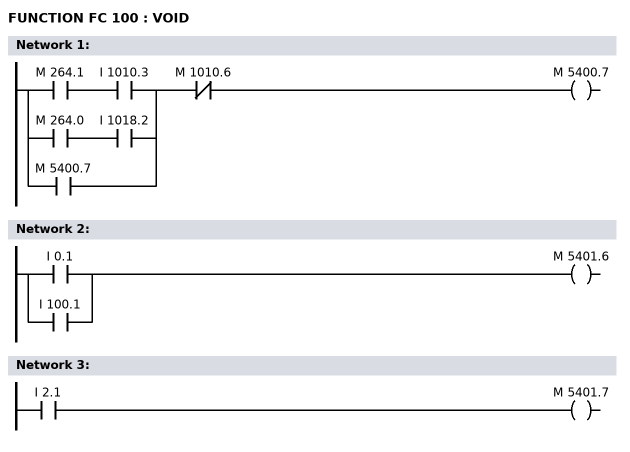

      A(    ;
      A     M    264.1;
      A     I   1010.3;
      O     ;
      A     M    264.0;
      A     I   1018.2;
      O     M   5400.7;
      )     ;
      AN    M   1010.6;
      =     M   5400.7;
NETWORK
TITLE =

      O     I      0.1;
      O     I    100.1;
      =     M   5401.6;
NETWORK
TITLE =

      A     I      2.1;
      =     M   5401.7;
NETWORK
TITLE =

      AN    OV;
      =     L      0.0;
      A     L      0.0;
      A     M   1003.7;
      AN    M   1000.0;
      A     M      0.5;
      =     M   5403.0;
      A     L      0.0;
      A     M   1003.7;
      A     M   1000.0;
      A     M      0.5;
      =     M   5403.1;
NETWORK
TITLE =

      AN    OV;
      =     L      0.0;
      A     L      0.0;
      A     M   1020.2;
      AN    I   1019.0;
      =     M   5403.2;
      A     L      0.0;
      A(    ;
      A     M   1020.2;
      A     I   1019.0;
      O     M   1035.1;
      )     ;
      =     M   5403.3;
NETWORK
TITLE =

      AN    OV;
      =     L      0.0;
      A     L      0.0;
      A     M   1008.2;
      AN    I   1011.0;
      =     M   5403.4;
      A     L      0.0;
      A(    ;
      A     M   1008.2;
      A     I   1011.0;
      O     M   1035.0;
      )     ;
      =     M   5403.5;
NETWORK
TITLE =
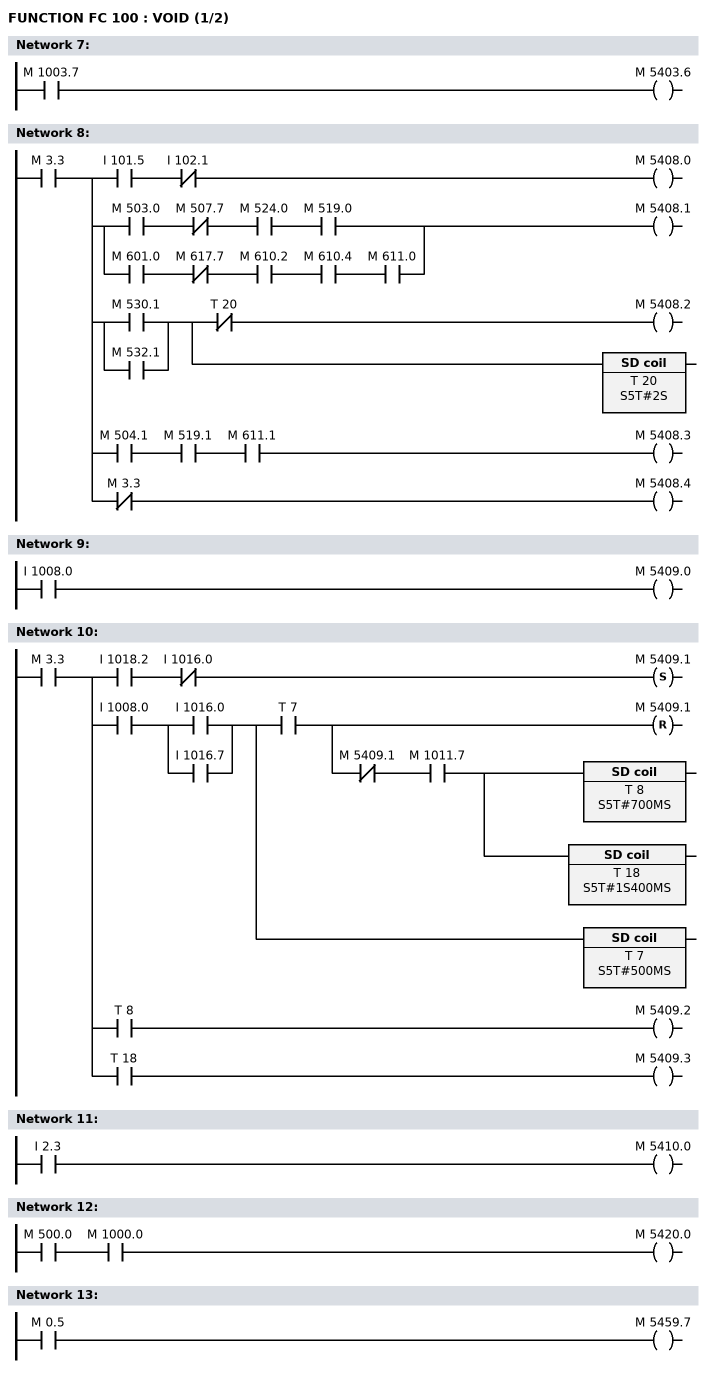

      A     M   1003.7;
      =     M   5403.6;
NETWORK
TITLE =

      A     M      3.3;
      =     L      0.0;
      A     L      0.0;
      A     I    101.5;
      AN    I    102.1;
      =     M   5408.0;
      A     L      0.0;
      A(    ;
      A     M    503.0;
      AN    M    507.7;
      A     M    524.0;
      A     M    519.0;
      O     ;
      A     M    601.0;
      AN    M    617.7;
      A     M    610.2;
      A     M    610.4;
      A     M    611.0;
      )     ;
      =     M   5408.1;
      A     L      0.0;
      A(    ;
      O     M    530.1;
      O     M    532.1;
      )     ;
      =     L      0.1;
      A     L      0.1;
      AN    T     20;
      =     M   5408.2;
      A     L      0.1;
      BLD   102;
      L     S5T#2S;
      SD    T     20;
      A     L      0.0;
      A     M    504.1;
      A     M    519.1;
      A     M    611.1;
      =     M   5408.3;
      A     L      0.0;
      AN    M      3.3;
      =     M   5408.4;
NETWORK
TITLE =

      A     I   1008.0;
      =     M   5409.0;
NETWORK
TITLE =

      A     M      3.3;
      =     L      0.0;
      A     L      0.0;
      A     I   1018.2;
      AN    I   1016.0;
      S     M   5409.1;
      A     L      0.0;
      A     I   1008.0;
      A(    ;
      O     I   1016.0;
      O     I   1016.7;
      )     ;
      =     L      0.1;
      A     L      0.1;
      A     T      7;
      =     L      0.2;
      A     L      0.2;
      BLD   102;
      R     M   5409.1;
      A     L      0.2;
      AN    M   5409.1;
      A     M   1011.7;
      L     S5T#700MS;
      SD    T      8;
      L     S5T#1S400MS;
      SD    T     18;
      A     L      0.1;
      BLD   102;
      L     S5T#500MS;
      SD    T      7;
      A     L      0.0;
      A     T      8;
      =     M   5409.2;
      A     L      0.0;
      A     T     18;
      =     M   5409.3;
NETWORK
TITLE =

      A     I      2.3;
      =     M   5410.0;
NETWORK
TITLE =

      A     M    500.0;
      A     M   1000.0;
      =     M   5420.0;
NETWORK
TITLE =

      A     M      0.5;
      =     M   5459.7;
NETWORK
TITLE =
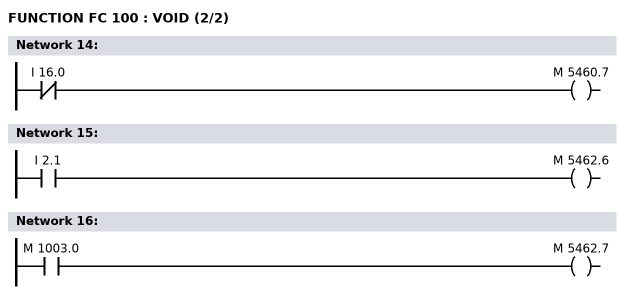

      AN    I     16.0;
      =     M   5460.7;
NETWORK
TITLE =

      A     I      2.1;
      =     M   5462.6;
NETWORK
TITLE =

      A     M   1003.0;
      =     M   5462.7;
NETWORK
TITLE =

      AN    OV;
      =     L      0.0;
      A     L      0.0;
      A(    ;
      ON    M    500.0;
      ON    I   1003.0;
      )     ;
      =     M   5463.0;
      A     L      0.0;
      A(    ;
      ON    M    500.6;
      ON    I   1000.4;
      )     ;
      =     M   5463.1;
      A     L      0.0;
      AN    M    516.0;
      AN    M    516.1;
      AN    M    516.2;
      AN    M    516.3;
      AN    M    516.4;
      AN    M    516.5;
      AN    M    516.6;
      AN    M    516.7;
      AN    M    517.1;
      AN    M    517.2;
      AN    M    517.3;
      AN    M   6060.0;
      AN    M    609.7;
      NOT   ;
      =     M   5463.2;
      A     L      0.0;
      A     M    517.0;
      =     M   5463.3;
      A     L      0.0;
      AN    M    541.0;
      AN    M    541.1;
      AN    M    543.0;
      NOT   ;
      =     M   5463.4;
      A     L      0.0;
      A     I    100.6;
      =     M   5463.5;
NETWORK
TITLE =

      AN    OV;
      =     L      0.0;
      A     L      0.0;
      AN    I   1011.0;
      =     M   5467.0;
      A     L      0.0;
      A     I   1011.1;
      =     M   5467.1;
      A     L      0.0;
      A     I   1011.2;
      =     M   5467.2;
      A     L      0.0;
      A     I   1011.4;
      =     M   5467.3;
      A     L      0.0;
      AN    M   1000.6;
      =     M   5467.4;
      A     L      0.0;
      A     I   1011.7;
      =     M   5467.6;
      A     L      0.0;
      A     M   1050.7;
      =     M   5467.7;
NETWORK
TITLE =
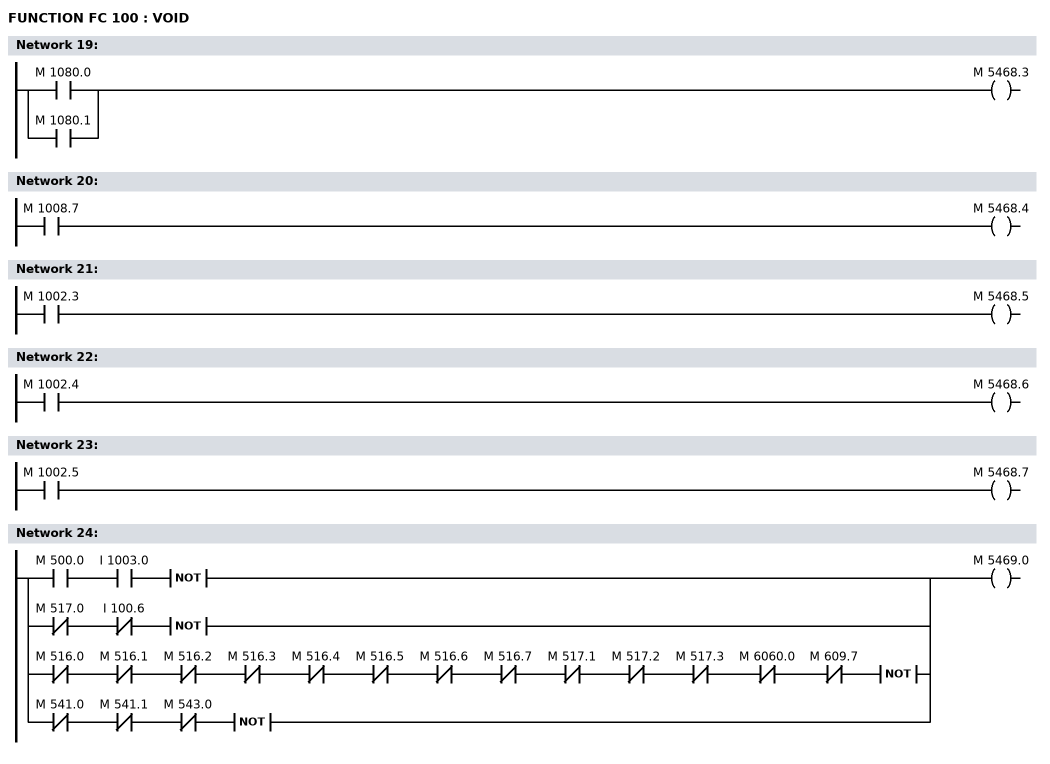

      O     M   1080.0;
      O     M   1080.1;
      =     M   5468.3;
NETWORK
TITLE =

      A     M   1008.7;
      =     M   5468.4;
NETWORK
TITLE =

      A     M   1002.3;
      =     M   5468.5;
NETWORK
TITLE =

      A     M   1002.4;
      =     M   5468.6;
NETWORK
TITLE =

      A     M   1002.5;
      =     M   5468.7;
NETWORK
TITLE =

      A     M    500.0;
      A     I   1003.0;
      NOT   ;
      O(    ;
      AN    M    517.0;
      AN    I    100.6;
      NOT   ;
      )     ;
      O(    ;
      AN    M    516.0;
      AN    M    516.1;
      AN    M    516.2;
      AN    M    516.3;
      AN    M    516.4;
      AN    M    516.5;
      AN    M    516.6;
      AN    M    516.7;
      AN    M    517.1;
      AN    M    517.2;
      AN    M    517.3;
      AN    M   6060.0;
      AN    M    609.7;
      NOT   ;
      )     ;
      O(    ;
      AN    M    541.0;
      AN    M    541.1;
      AN    M    543.0;
      NOT   ;
      )     ;
      =     M   5469.0;
END_FUNCTION

FUNCTION FC 101 : VOID
TITLE =
VERSION : 0.1

BEGIN
NETWORK
TITLE =
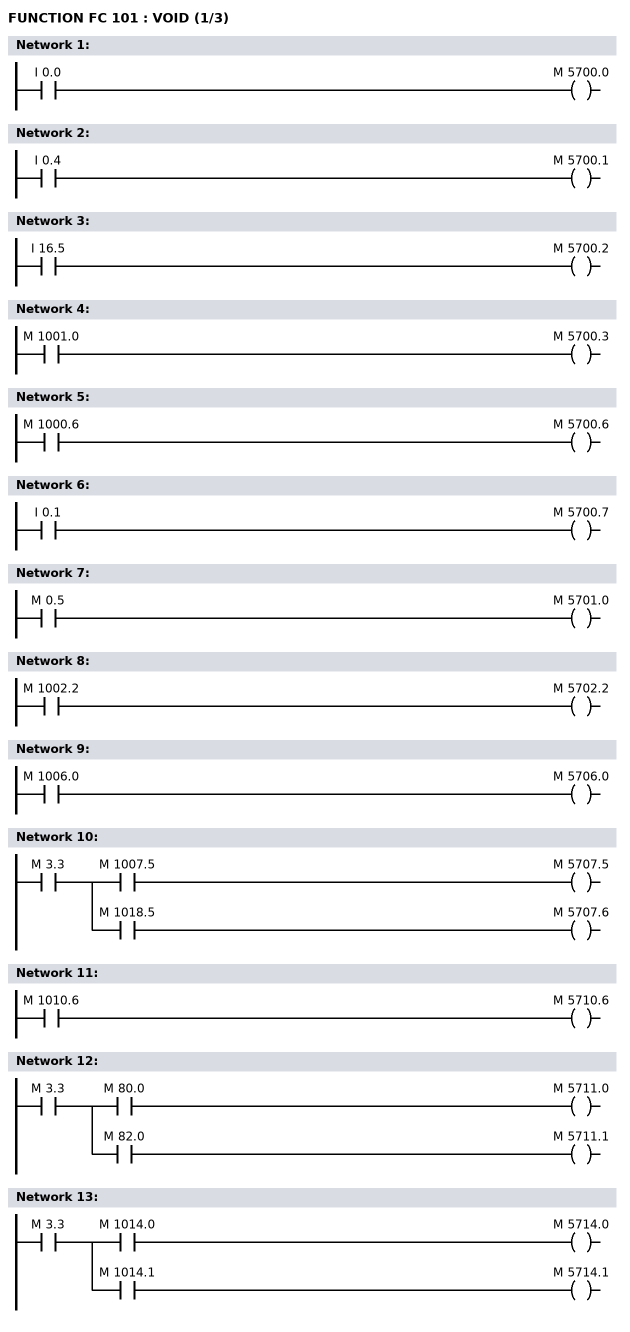

      A     I      0.0;
      =     M   5700.0;
NETWORK
TITLE =

      A     I      0.4;
      =     M   5700.1;
NETWORK
TITLE =

      A     I     16.5;
      =     M   5700.2;
NETWORK
TITLE =

      A     M   1001.0;
      =     M   5700.3;
NETWORK
TITLE =

      A     M   1000.6;
      =     M   5700.6;
NETWORK
TITLE =

      A     I      0.1;
      =     M   5700.7;
NETWORK
TITLE =

      A     M      0.5;
      =     M   5701.0;
NETWORK
TITLE =

      A     M   1002.2;
      =     M   5702.2;
NETWORK
TITLE =

      A     M   1006.0;
      =     M   5706.0;
NETWORK
TITLE =

      A     M      3.3;
      =     L      0.0;
      A     L      0.0;
      A     M   1007.5;
      =     M   5707.5;
      A     L      0.0;
      A     M   1018.5;
      =     M   5707.6;
NETWORK
TITLE =

      A     M   1010.6;
      =     M   5710.6;
NETWORK
TITLE =

      A     M      3.3;
      =     L      0.0;
      A     L      0.0;
      A     M     80.0;
      =     M   5711.0;
      A     L      0.0;
      A     M     82.0;
      =     M   5711.1;
NETWORK
TITLE =

      A     M      3.3;
      =     L      0.0;
      A     L      0.0;
      A     M   1014.0;
      =     M   5714.0;
      A     L      0.0;
      A     M   1014.1;
      =     M   5714.1;
NETWORK
TITLE =
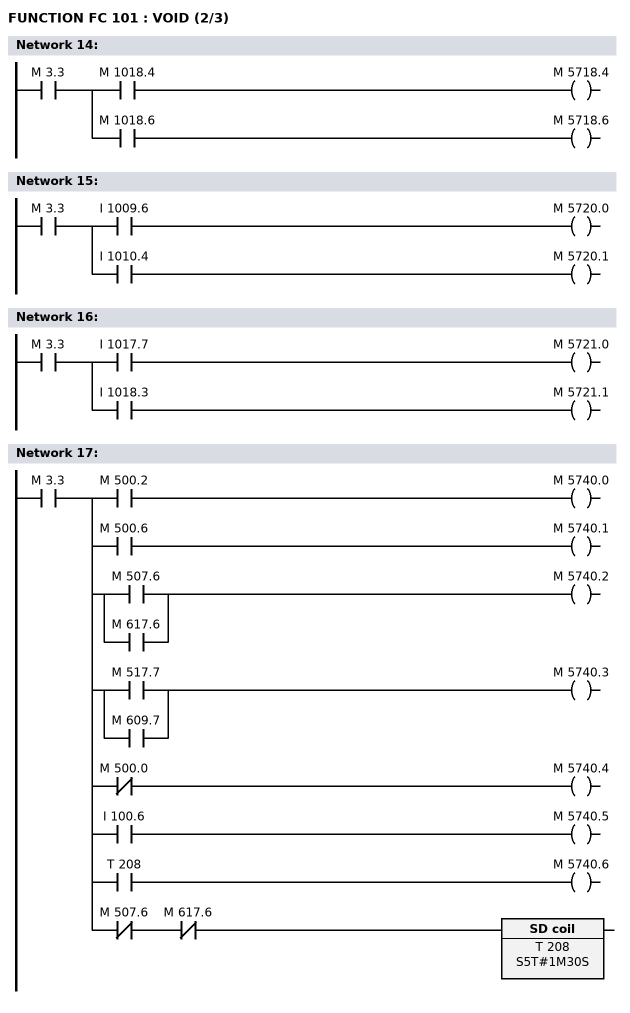

      A     M      3.3;
      =     L      0.0;
      A     L      0.0;
      A     M   1018.4;
      =     M   5718.4;
      A     L      0.0;
      A     M   1018.6;
      =     M   5718.6;
NETWORK
TITLE =

      A     M      3.3;
      =     L      0.0;
      A     L      0.0;
      A     I   1009.6;
      =     M   5720.0;
      A     L      0.0;
      A     I   1010.4;
      =     M   5720.1;
NETWORK
TITLE =

      A     M      3.3;
      =     L      0.0;
      A     L      0.0;
      A     I   1017.7;
      =     M   5721.0;
      A     L      0.0;
      A     I   1018.3;
      =     M   5721.1;
NETWORK
TITLE =

      A     M      3.3;
      =     L      0.0;
      A     L      0.0;
      A     M    500.2;
      =     M   5740.0;
      A     L      0.0;
      A     M    500.6;
      =     M   5740.1;
      A     L      0.0;
      A(    ;
      O     M    507.6;
      O     M    617.6;
      )     ;
      =     M   5740.2;
      A     L      0.0;
      A(    ;
      O     M    517.7;
      O     M    609.7;
      )     ;
      =     M   5740.3;
      A     L      0.0;
      AN    M    500.0;
      =     M   5740.4;
      A     L      0.0;
      A     I    100.6;
      =     M   5740.5;
      A     L      0.0;
      A     T    208;
      =     M   5740.6;
      A     L      0.0;
      AN    M    507.6;
      AN    M    617.6;
      L     S5T#1M30S;
      SD    T    208;
NETWORK
TITLE =
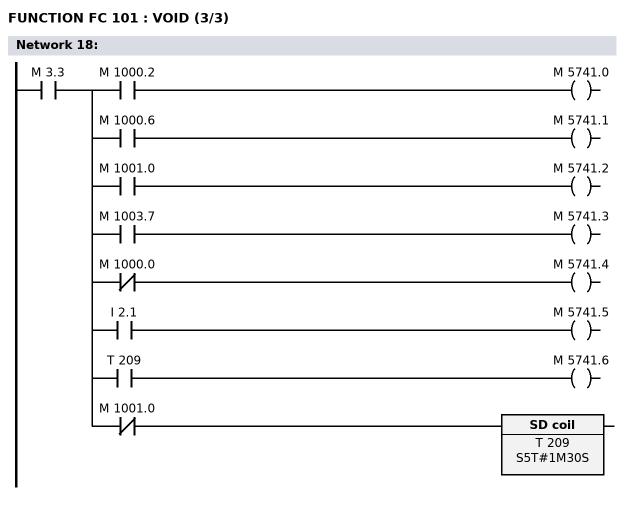

      A     M      3.3;
      =     L      0.0;
      A     L      0.0;
      A     M   1000.2;
      =     M   5741.0;
      A     L      0.0;
      A     M   1000.6;
      =     M   5741.1;
      A     L      0.0;
      A     M   1001.0;
      =     M   5741.2;
      A     L      0.0;
      A     M   1003.7;
      =     M   5741.3;
      A     L      0.0;
      AN    M   1000.0;
      =     M   5741.4;
      A     L      0.0;
      A     I      2.1;
      =     M   5741.5;
      A     L      0.0;
      A     T    209;
      =     M   5741.6;
      A     L      0.0;
      AN    M   1001.0;
      L     S5T#1M30S;
      SD    T    209;
END_FUNCTION

FUNCTION_BLOCK FB 105
TITLE =
VERSION : 0.1


VAR
  S711A_RBT1_WELD_OK_PLS : BOOL ;
  S711A_RBT1_WELD_NG_PLS : BOOL ;
  S711A_RBT1_WELD_PASS_PLS : BOOL ;
  S711A_CHECK_SUM_PLS : BOOL ;
  S711A_WELD_DATA_MOV_BUFF : BOOL ;
  MW_0_BUFF : ARRAY  [0 .. 59 ] OF WORD ;
  PLS1 : BOOL ;
  PLS2 : BOOL ;
END_VAR
VAR_TEMP
  SFC20_RET_VAL : INT ;
END_VAR
BEGIN
NETWORK
TITLE =MES 용접누락 DATA -> #711A차종코드(2011) 기준값 버퍼로 전송(LM)
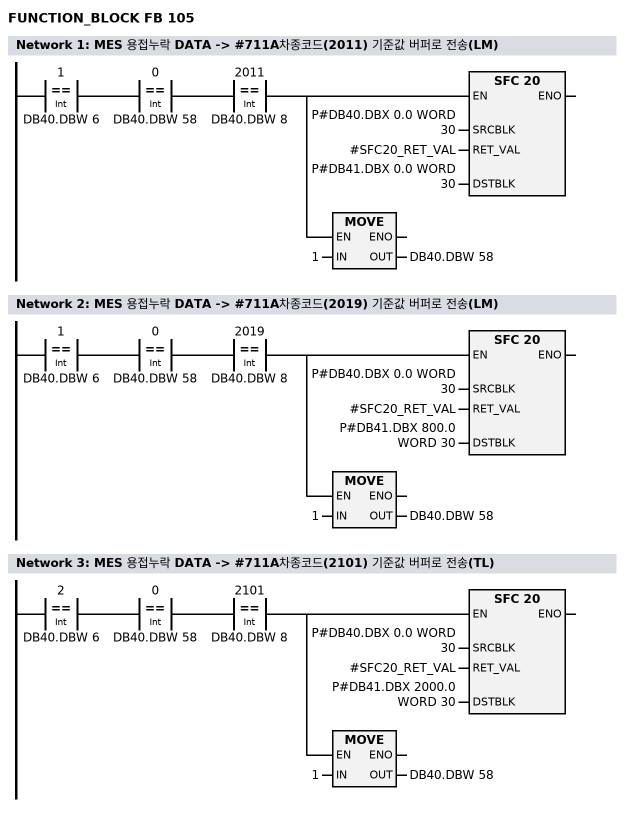

      A(    ;
      L     1;
      L     DB40.DBW    6;
      ==I   ;
      )     ;
      A(    ;
      L     0;
      L     DB40.DBW   58;
      ==I   ;
      )     ;
      A(    ;
      L     2011;
      L     DB40.DBW    8;
      ==I   ;
      )     ;
      =     L      2.0;
      A     L      2.0;
      JNB   _001;
      CALL SFC   20 (
           SRCBLK                   := P#DB40.DBX 0.0 WORD 30,
           RET_VAL                  := #SFC20_RET_VAL,
           DSTBLK                   := P#DB41.DBX 0.0 WORD 30);
_001: NOP   0;
      A     L      2.0;
      JNB   _002;
      L     1;
      T     DB40.DBW   58;
_002: NOP   0;
NETWORK
TITLE =MES 용접누락 DATA -> #711A차종코드(2019) 기준값 버퍼로 전송(LM)

      A(    ;
      L     1;
      L     DB40.DBW    6;
      ==I   ;
      )     ;
      A(    ;
      L     0;
      L     DB40.DBW   58;
      ==I   ;
      )     ;
      A(    ;
      L     2019;
      L     DB40.DBW    8;
      ==I   ;
      )     ;
      =     L      2.0;
      A     L      2.0;
      JNB   _003;
      CALL SFC   20 (
           SRCBLK                   := P#DB40.DBX 0.0 WORD 30,
           RET_VAL                  := #SFC20_RET_VAL,
           DSTBLK                   := P#DB41.DBX 800.0 WORD 30);
_003: NOP   0;
      A     L      2.0;
      JNB   _004;
      L     1;
      T     DB40.DBW   58;
_004: NOP   0;
NETWORK
TITLE =MES 용접누락 DATA -> #711A차종코드(2101) 기준값 버퍼로 전송(TL)

      A(    ;
      L     2;
      L     DB40.DBW    6;
      ==I   ;
      )     ;
      A(    ;
      L     0;
      L     DB40.DBW   58;
      ==I   ;
      )     ;
      A(    ;
      L     2101;
      L     DB40.DBW    8;
      ==I   ;
      )     ;
      =     L      2.0;
      A     L      2.0;
      JNB   _005;
      CALL SFC   20 (
           SRCBLK                   := P#DB40.DBX 0.0 WORD 30,
           RET_VAL                  := #SFC20_RET_VAL,
           DSTBLK                   := P#DB41.DBX 2000.0 WORD 30);
_005: NOP   0;
      A     L      2.0;
      JNB   _006;
      L     1;
      T     DB40.DBW   58;
_006: NOP   0;
NETWORK
TITLE =#711A-2 RBT1호 용접카운터 INT -> DB로 전송보조

      AN    OV;
      =     L      2.0;
      A     L      2.0;
      A     I   1004.0;
      =     M     11.0;
      A     L      2.0;
      A     I   1004.1;
      =     M     11.1;
      A     L      2.0;
      A     I   1004.2;
      =     M     11.2;
      A     L      2.0;
      A     I   1004.3;
      =     M     11.3;
      A     L      2.0;
      A     I   1004.4;
      =     M     11.4;
      A     L      2.0;
      AN    M      3.3;
      =     L      2.1;
      A     L      2.1;
      A     I   1004.5;
      =     M     11.5;
      A     L      2.1;
      A     I   1004.6;
      =     M     11.6;
      A     L      2.1;
      A     I   1004.7;
      =     M     11.7;
      A     L      2.0;
      AN    I    102.1;
      A     I   1000.1;
      S     M    531.7;
      A     L      2.0;
      AN    I    102.1;
      A     M    505.1;
      A     M    540.1;
      A     M    540.7;
      R     M    531.7;
NETWORK
TITLE =#711A-2 RBT1호 용접카운터 INT -> DB로 전송
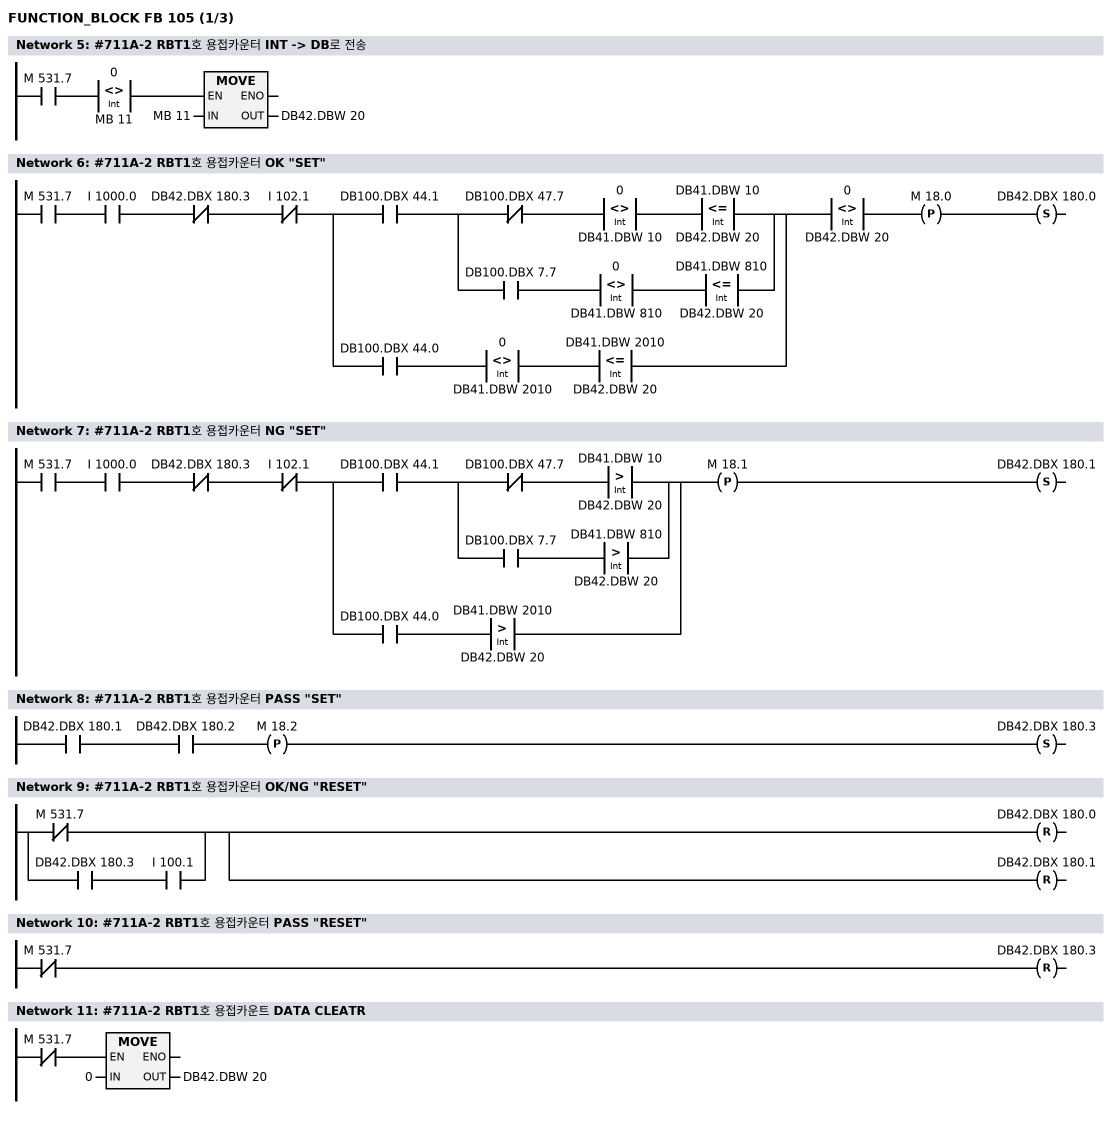

      A     M    531.7;
      A(    ;
      L     0;
      L     MB    11;
      <>I   ;
      )     ;
      JNB   _007;
      L     MB    11;
      T     DB42.DBW   20;
_007: NOP   0;
NETWORK
TITLE =#711A-2 RBT1호 용접카운터 OK "SET"

      A     M    531.7;
      A     I   1000.0;
      AN    DB42.DBX  180.3;
      AN    I    102.1;
      A(    ;
      A     DB100.DBX   44.1;
      A(    ;
      AN    DB100.DBX   47.7;
      A(    ;
      L     0;
      L     DB41.DBW   10;
      <>I   ;
      )     ;
      A(    ;
      L     DB41.DBW   10;
      L     DB42.DBW   20;
      <=I   ;
      )     ;
      O     ;
      A     DB100.DBX    7.7;
      A(    ;
      L     0;
      L     DB41.DBW  810;
      <>I   ;
      )     ;
      A(    ;
      L     DB41.DBW  810;
      L     DB42.DBW   20;
      <=I   ;
      )     ;
      )     ;
      O     ;
      A     DB100.DBX   44.0;
      A(    ;
      L     0;
      L     DB41.DBW 2010;
      <>I   ;
      )     ;
      A(    ;
      L     DB41.DBW 2010;
      L     DB42.DBW   20;
      <=I   ;
      )     ;
      )     ;
      A(    ;
      L     0;
      L     DB42.DBW   20;
      <>I   ;
      )     ;
      FP    M     18.0;
      S     DB42.DBX  180.0;
NETWORK
TITLE =#711A-2 RBT1호 용접카운터 NG "SET"

      A     M    531.7;
      A     I   1000.0;
      AN    DB42.DBX  180.3;
      AN    I    102.1;
      A(    ;
      A     DB100.DBX   44.1;
      A(    ;
      AN    DB100.DBX   47.7;
      A(    ;
      L     DB41.DBW   10;
      L     DB42.DBW   20;
      >I    ;
      )     ;
      O     ;
      A     DB100.DBX    7.7;
      A(    ;
      L     DB41.DBW  810;
      L     DB42.DBW   20;
      >I    ;
      )     ;
      )     ;
      O     ;
      A     DB100.DBX   44.0;
      A(    ;
      L     DB41.DBW 2010;
      L     DB42.DBW   20;
      >I    ;
      )     ;
      )     ;
      FP    M     18.1;
      S     DB42.DBX  180.1;
NETWORK
TITLE =#711A-2 RBT1호 용접카운터 PASS "SET"

      A     DB42.DBX  180.1;
      A     DB42.DBX  180.2;
      FP    M     18.2;
      S     DB42.DBX  180.3;
NETWORK
TITLE =#711A-2 RBT1호 용접카운터 OK/NG "RESET"

      ON    M    531.7;
      O     ;
      A     DB42.DBX  180.3;
      A     I    100.1;
      R     DB42.DBX  180.0;
      R     DB42.DBX  180.1;
NETWORK
TITLE =#711A-2 RBT1호 용접카운터 PASS "RESET"

      AN    M    531.7;
      R     DB42.DBX  180.3;
NETWORK
TITLE =#711A-2 RBT1호 용접카운트 DATA CLEATR

      AN    M    531.7;
      JNB   _008;
      L     0;
      T     DB42.DBW   20;
_008: NOP   0;
NETWORK
TITLE =#711A-2 RBT1호 용접DATA 관련(공정 및 차종정보)
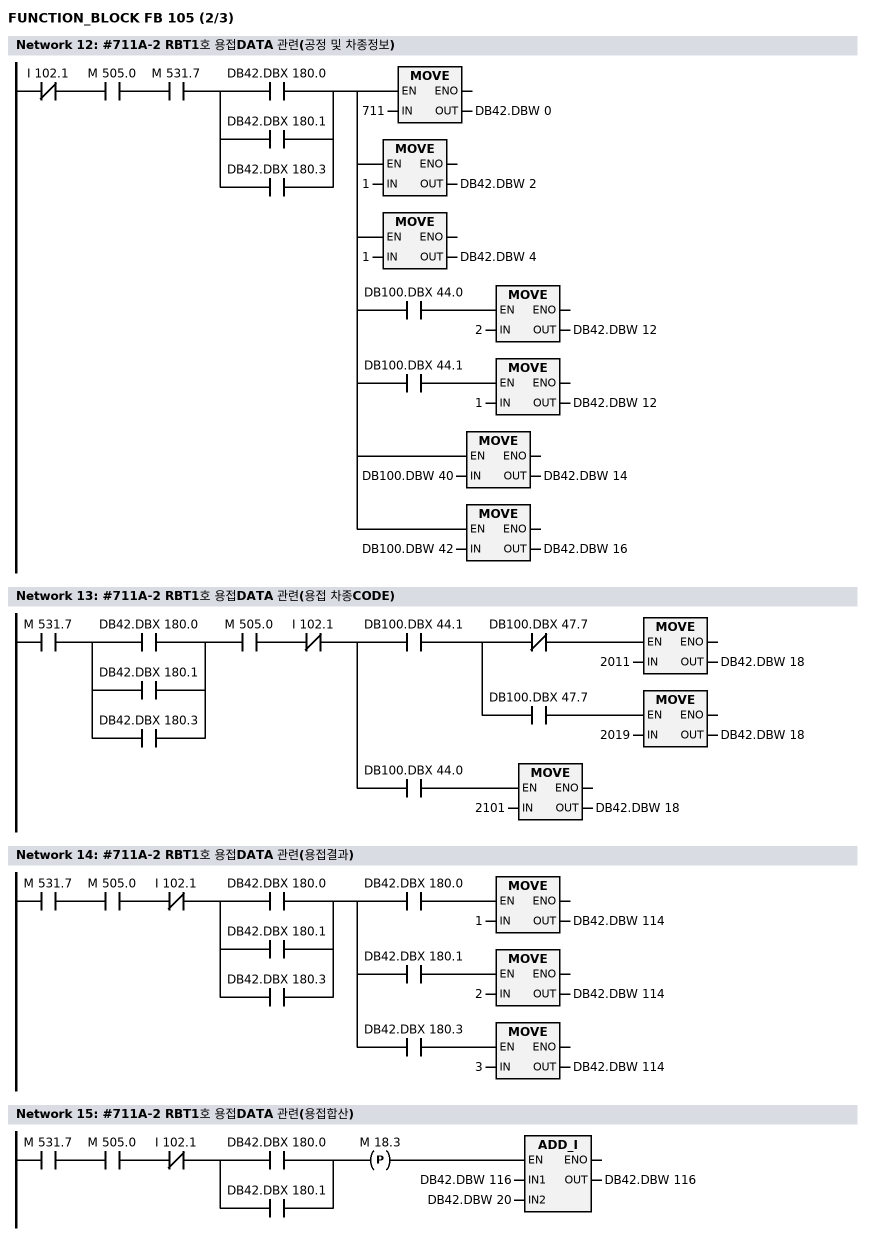

      AN    I    102.1;
      A     M    505.0;
      A     M    531.7;
      A(    ;
      O     DB42.DBX  180.0;
      O     DB42.DBX  180.1;
      O     DB42.DBX  180.3;
      )     ;
      =     L      2.0;
      A     L      2.0;
      JNB   _009;
      L     711;
      T     DB42.DBW    0;
_009: NOP   0;
      A     L      2.0;
      JNB   _00a;
      L     1;
      T     DB42.DBW    2;
_00a: NOP   0;
      A     L      2.0;
      JNB   _00b;
      L     1;
      T     DB42.DBW    4;
_00b: NOP   0;
      A     L      2.0;
      A     DB100.DBX   44.0;
      JNB   _00c;
      L     2;
      T     DB42.DBW   12;
_00c: NOP   0;
      A     L      2.0;
      A     DB100.DBX   44.1;
      JNB   _00d;
      L     1;
      T     DB42.DBW   12;
_00d: NOP   0;
      A     L      2.0;
      JNB   _00e;
      L     DB100.DBW   40;
      T     DB42.DBW   14;
_00e: NOP   0;
      A     L      2.0;
      JNB   _00f;
      L     DB100.DBW   42;
      T     DB42.DBW   16;
_00f: NOP   0;
NETWORK
TITLE =#711A-2 RBT1호 용접DATA 관련(용접 차종CODE)

      A     M    531.7;
      A(    ;
      O     DB42.DBX  180.0;
      O     DB42.DBX  180.1;
      O     DB42.DBX  180.3;
      )     ;
      A     M    505.0;
      AN    I    102.1;
      =     L      2.0;
      A     L      2.0;
      A     DB100.DBX   44.1;
      =     L      2.1;
      A     L      2.1;
      AN    DB100.DBX   47.7;
      JNB   _010;
      L     2011;
      T     DB42.DBW   18;
_010: NOP   0;
      A     L      2.1;
      A     DB100.DBX   47.7;
      JNB   _011;
      L     2019;
      T     DB42.DBW   18;
_011: NOP   0;
      A     L      2.0;
      A     DB100.DBX   44.0;
      JNB   _012;
      L     2101;
      T     DB42.DBW   18;
_012: NOP   0;
NETWORK
TITLE =#711A-2 RBT1호 용접DATA 관련(용접결과)

      A     M    531.7;
      A     M    505.0;
      AN    I    102.1;
      A(    ;
      O     DB42.DBX  180.0;
      O     DB42.DBX  180.1;
      O     DB42.DBX  180.3;
      )     ;
      =     L      2.0;
      A     L      2.0;
      A     DB42.DBX  180.0;
      JNB   _013;
      L     1;
      T     DB42.DBW  114;
_013: NOP   0;
      A     L      2.0;
      A     DB42.DBX  180.1;
      JNB   _014;
      L     2;
      T     DB42.DBW  114;
_014: NOP   0;
      A     L      2.0;
      A     DB42.DBX  180.3;
      JNB   _015;
      L     3;
      T     DB42.DBW  114;
_015: NOP   0;
NETWORK
TITLE =#711A-2 RBT1호 용접DATA 관련(용접합산)

      A     M    531.7;
      A     M    505.0;
      AN    I    102.1;
      A(    ;
      O     DB42.DBX  180.0;
      O     DB42.DBX  180.1;
      )     ;
      FP    M     18.3;
      JNB   _016;
      L     DB42.DBW  116;
      L     DB42.DBW   20;
      +I    ;
      T     DB42.DBW  116;
_016: NOP   0;
NETWORK
TITLE =용접누락버퍼로 공정DATA 전송
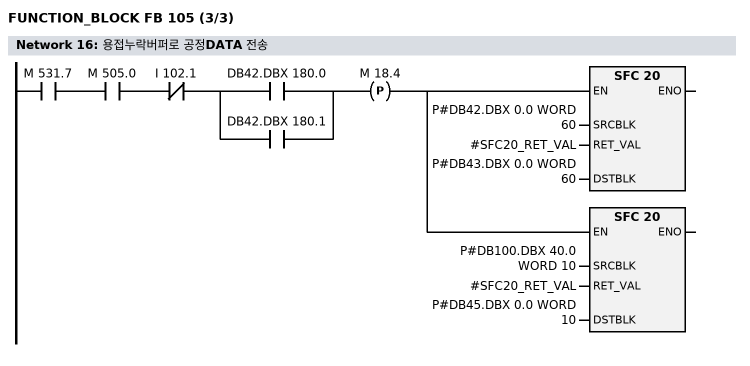

      A     M    531.7;
      A     M    505.0;
      AN    I    102.1;
      A(    ;
      O     DB42.DBX  180.0;
      O     DB42.DBX  180.1;
      )     ;
      FP    M     18.4;
      =     L      2.0;
      A     L      2.0;
      JNB   _017;
      CALL SFC   20 (
           SRCBLK                   := P#DB42.DBX 0.0 WORD 60,
           RET_VAL                  := #SFC20_RET_VAL,
           DSTBLK                   := P#DB43.DBX 0.0 WORD 60);
_017: NOP   0;
      A     L      2.0;
      JNB   _018;
      CALL SFC   20 (
           SRCBLK                   := P#DB100.DBX 40.0 WORD 10,
           RET_VAL                  := #SFC20_RET_VAL,
           DSTBLK                   := P#DB45.DBX 0.0 WORD 10);
_018: NOP   0;
NETWORK
TITLE =용접누락버퍼로 공정DATA 전송

      AN    M    531.7;
      FP    M     18.5;
      =     L      2.0;
      A(    ;
      A     L      2.0;
      JNB   _019;
      CALL SFC   20 (
           SRCBLK                   := P#DB43.DBX 960.0 WORD 60,
           RET_VAL                  := #SFC20_RET_VAL,
           DSTBLK                   := P#DB43.DBX 1080.0 WORD 60);
_019: A     BR;
      )     ;
      JNB   _01a;
      CALL SFC   20 (
           SRCBLK                   := P#DB43.DBX 840.0 WORD 60,
           RET_VAL                  := #SFC20_RET_VAL,
           DSTBLK                   := P#DB43.DBX 960.0 WORD 60);
_01a: NOP   0;
      A(    ;
      A     L      2.0;
      JNB   _01b;
      CALL SFC   20 (
           SRCBLK                   := P#DB43.DBX 720.0 WORD 60,
           RET_VAL                  := #SFC20_RET_VAL,
           DSTBLK                   := P#DB43.DBX 840.0 WORD 60);
_01b: A     BR;
      )     ;
      JNB   _01c;
      CALL SFC   20 (
           SRCBLK                   := P#DB43.DBX 600.0 WORD 60,
           RET_VAL                  := #SFC20_RET_VAL,
           DSTBLK                   := P#DB43.DBX 720.0 WORD 60);
_01c: NOP   0;
      A(    ;
      A     L      2.0;
      JNB   _01d;
      CALL SFC   20 (
           SRCBLK                   := P#DB43.DBX 480.0 WORD 60,
           RET_VAL                  := #SFC20_RET_VAL,
           DSTBLK                   := P#DB43.DBX 600.0 WORD 60);
_01d: A     BR;
      )     ;
      JNB   _01e;
      CALL SFC   20 (
           SRCBLK                   := P#DB43.DBX 360.0 WORD 60,
           RET_VAL                  := #SFC20_RET_VAL,
           DSTBLK                   := P#DB43.DBX 480.0 WORD 60);
_01e: NOP   0;
      A(    ;
      A     L      2.0;
      JNB   _01f;
      CALL SFC   20 (
           SRCBLK                   := P#DB43.DBX 240.0 WORD 60,
           RET_VAL                  := #SFC20_RET_VAL,
           DSTBLK                   := P#DB43.DBX 360.0 WORD 60);
_01f: A     BR;
      )     ;
      JNB   _020;
      CALL SFC   20 (
           SRCBLK                   := P#DB43.DBX 120.0 WORD 60,
           RET_VAL                  := #SFC20_RET_VAL,
           DSTBLK                   := P#DB43.DBX 240.0 WORD 60);
_020: NOP   0;
      A     L      2.0;
      JNB   _021;
      CALL SFC   20 (
           SRCBLK                   := P#DB43.DBX 0.0 WORD 60,
           RET_VAL                  := #SFC20_RET_VAL,
           DSTBLK                   := P#DB43.DBX 120.0 WORD 60);
_021: NOP   0;
      A     L      2.0;
      JNB   _022;
      CALL SFC   21 (
           BVAL                     := P#M 30.0 WORD 1,
           RET_VAL                  := #SFC20_RET_VAL,
           BLK                      := P#DB43.DBX 0.0 WORD 60);
_022: NOP   0;
      A(    ;
      A     L      2.0;
      JNB   _023;
      CALL SFC   20 (
           SRCBLK                   := P#DB45.DBX 160.0 WORD 10,
           RET_VAL                  := #SFC20_RET_VAL,
           DSTBLK                   := P#DB45.DBX 180.0 WORD 10);
_023: A     BR;
      )     ;
      JNB   _024;
      CALL SFC   20 (
           SRCBLK                   := P#DB45.DBX 140.0 WORD 10,
           RET_VAL                  := #SFC20_RET_VAL,
           DSTBLK                   := P#DB45.DBX 160.0 WORD 10);
_024: NOP   0;
      A(    ;
      A     L      2.0;
      JNB   _025;
      CALL SFC   20 (
           SRCBLK                   := P#DB45.DBX 120.0 WORD 10,
           RET_VAL                  := #SFC20_RET_VAL,
           DSTBLK                   := P#DB45.DBX 140.0 WORD 10);
_025: A     BR;
      )     ;
      JNB   _026;
      CALL SFC   20 (
           SRCBLK                   := P#DB45.DBX 100.0 WORD 10,
           RET_VAL                  := #SFC20_RET_VAL,
           DSTBLK                   := P#DB45.DBX 120.0 WORD 10);
_026: NOP   0;
      A(    ;
      A     L      2.0;
      JNB   _027;
      CALL SFC   20 (
           SRCBLK                   := P#DB45.DBX 80.0 WORD 10,
           RET_VAL                  := #SFC20_RET_VAL,
           DSTBLK                   := P#DB45.DBX 100.0 WORD 10);
_027: A     BR;
      )     ;
      JNB   _028;
      CALL SFC   20 (
           SRCBLK                   := P#DB45.DBX 60.0 WORD 10,
           RET_VAL                  := #SFC20_RET_VAL,
           DSTBLK                   := P#DB45.DBX 80.0 WORD 10);
_028: NOP   0;
      A(    ;
      A     L      2.0;
      JNB   _029;
      CALL SFC   20 (
           SRCBLK                   := P#DB45.DBX 40.0 WORD 10,
           RET_VAL                  := #SFC20_RET_VAL,
           DSTBLK                   := P#DB45.DBX 60.0 WORD 10);
_029: A     BR;
      )     ;
      JNB   _02a;
      CALL SFC   20 (
           SRCBLK                   := P#DB45.DBX 20.0 WORD 10,
           RET_VAL                  := #SFC20_RET_VAL,
           DSTBLK                   := P#DB45.DBX 40.0 WORD 10);
_02a: NOP   0;
      A     L      2.0;
      JNB   _02b;
      CALL SFC   20 (
           SRCBLK                   := P#DB45.DBX 0.0 WORD 10,
           RET_VAL                  := #SFC20_RET_VAL,
           DSTBLK                   := P#DB45.DBX 20.0 WORD 10);
_02b: NOP   0;
      A     L      2.0;
      JNB   _02c;
      CALL SFC   21 (
           BVAL                     := P#M 30.0 WORD 1,
           RET_VAL                  := #SFC20_RET_VAL,
           BLK                      := P#DB45.DBX 0.0 WORD 10);
_02c: NOP   0;
NETWORK
TITLE =용접누락버퍼로 공정DATA 전송
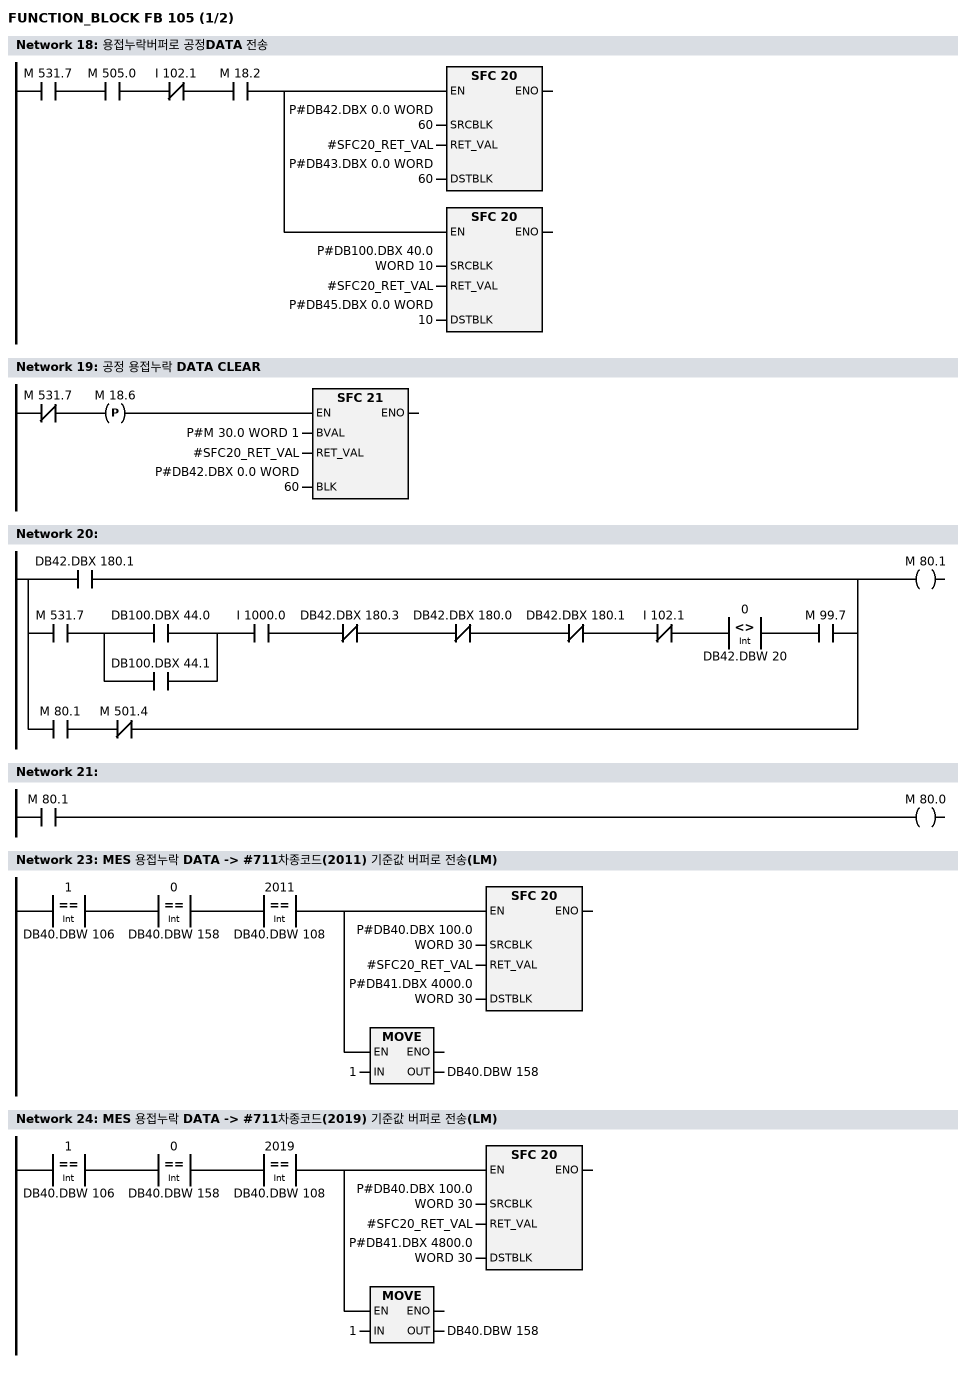

      A     M    531.7;
      A     M    505.0;
      AN    I    102.1;
      A     M     18.2;
      =     L      2.0;
      A     L      2.0;
      JNB   _02d;
      CALL SFC   20 (
           SRCBLK                   := P#DB42.DBX 0.0 WORD 60,
           RET_VAL                  := #SFC20_RET_VAL,
           DSTBLK                   := P#DB43.DBX 0.0 WORD 60);
_02d: NOP   0;
      A     L      2.0;
      JNB   _02e;
      CALL SFC   20 (
           SRCBLK                   := P#DB100.DBX 40.0 WORD 10,
           RET_VAL                  := #SFC20_RET_VAL,
           DSTBLK                   := P#DB45.DBX 0.0 WORD 10);
_02e: NOP   0;
NETWORK
TITLE =공정 용접누락 DATA CLEAR

      AN    M    531.7;
      FP    M     18.6;
      JNB   _02f;
      CALL SFC   21 (
           BVAL                     := P#M 30.0 WORD 1,
           RET_VAL                  := #SFC20_RET_VAL,
           BLK                      := P#DB42.DBX 0.0 WORD 60);
_02f: NOP   0;
NETWORK
TITLE =

      O     DB42.DBX  180.1;
      O     ;
      A     M    531.7;
      A(    ;
      O     DB100.DBX   44.0;
      O     DB100.DBX   44.1;
      )     ;
      A     I   1000.0;
      AN    DB42.DBX  180.3;
      AN    DB42.DBX  180.0;
      AN    DB42.DBX  180.1;
      AN    I    102.1;
      A(    ;
      L     0;
      L     DB42.DBW   20;
      <>I   ;
      )     ;
      A     M     99.7;
      O     ;
      A     M     80.1;
      AN    M    501.4;
      =     M     80.1;
NETWORK
TITLE =

      A     M     80.1;
      =     M     80.0;
NETWORK
TITLE =

NETWORK
TITLE =MES 용접누락 DATA -> #711차종코드(2011) 기준값 버퍼로 전송(LM)

      A(    ;
      L     1;
      L     DB40.DBW  106;
      ==I   ;
      )     ;
      A(    ;
      L     0;
      L     DB40.DBW  158;
      ==I   ;
      )     ;
      A(    ;
      L     2011;
      L     DB40.DBW  108;
      ==I   ;
      )     ;
      =     L      2.0;
      A     L      2.0;
      JNB   _030;
      CALL SFC   20 (
           SRCBLK                   := P#DB40.DBX 100.0 WORD 30,
           RET_VAL                  := #SFC20_RET_VAL,
           DSTBLK                   := P#DB41.DBX 4000.0 WORD 30);
_030: NOP   0;
      A     L      2.0;
      JNB   _031;
      L     1;
      T     DB40.DBW  158;
_031: NOP   0;
NETWORK
TITLE =MES 용접누락 DATA -> #711차종코드(2019) 기준값 버퍼로 전송(LM)

      A(    ;
      L     1;
      L     DB40.DBW  106;
      ==I   ;
      )     ;
      A(    ;
      L     0;
      L     DB40.DBW  158;
      ==I   ;
      )     ;
      A(    ;
      L     2019;
      L     DB40.DBW  108;
      ==I   ;
      )     ;
      =     L      2.0;
      A     L      2.0;
      JNB   _032;
      CALL SFC   20 (
           SRCBLK                   := P#DB40.DBX 100.0 WORD 30,
           RET_VAL                  := #SFC20_RET_VAL,
           DSTBLK                   := P#DB41.DBX 4800.0 WORD 30);
_032: NOP   0;
      A     L      2.0;
      JNB   _033;
      L     1;
      T     DB40.DBW  158;
_033: NOP   0;
NETWORK
TITLE =MES 용접누락 DATA -> #711차종코드(2101) 기준값 버퍼로 전송(TL)
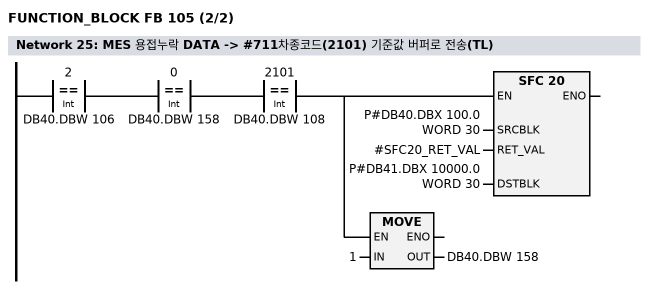

      A(    ;
      L     2;
      L     DB40.DBW  106;
      ==I   ;
      )     ;
      A(    ;
      L     0;
      L     DB40.DBW  158;
      ==I   ;
      )     ;
      A(    ;
      L     2101;
      L     DB40.DBW  108;
      ==I   ;
      )     ;
      =     L      2.0;
      A     L      2.0;
      JNB   _034;
      CALL SFC   20 (
           SRCBLK                   := P#DB40.DBX 100.0 WORD 30,
           RET_VAL                  := #SFC20_RET_VAL,
           DSTBLK                   := P#DB41.DBX 10000.0 WORD 30);
_034: NOP   0;
      A     L      2.0;
      JNB   _035;
      L     1;
      T     DB40.DBW  158;
_035: NOP   0;
NETWORK
TITLE =#711 RBT2호 용접카운터 INT -> DB로 전송보조

      AN    OV;
      =     L      2.0;
      A     L      2.0;
      A     I   1020.0;
      =     M     15.0;
      A     L      2.0;
      A     I   1020.1;
      =     M     15.1;
      A     L      2.0;
      A     I   1020.2;
      =     M     15.2;
      A     L      2.0;
      A     I   1020.3;
      =     M     15.3;
      A     L      2.0;
      A     I   1020.4;
      =     M     15.4;
      A     L      2.0;
      AN    M      3.3;
      =     L      2.1;
      A     L      2.1;
      A     I   1020.5;
      =     M     15.5;
      A     L      2.1;
      A     I   1020.6;
      =     M     15.6;
      A     L      2.1;
      A     I   1020.7;
      =     M     15.7;
      A     L      2.0;
      A     I   1016.1;
      S     M     16.7;
      A     L      2.0;
      A(    ;
      A     M   1010.7;
      A     M   1002.1;
      O     M   4712.1;
      )     ;
      R     M     16.7;
NETWORK
TITLE =#711 RBT2호 용접카운터 INT -> DB로 전송
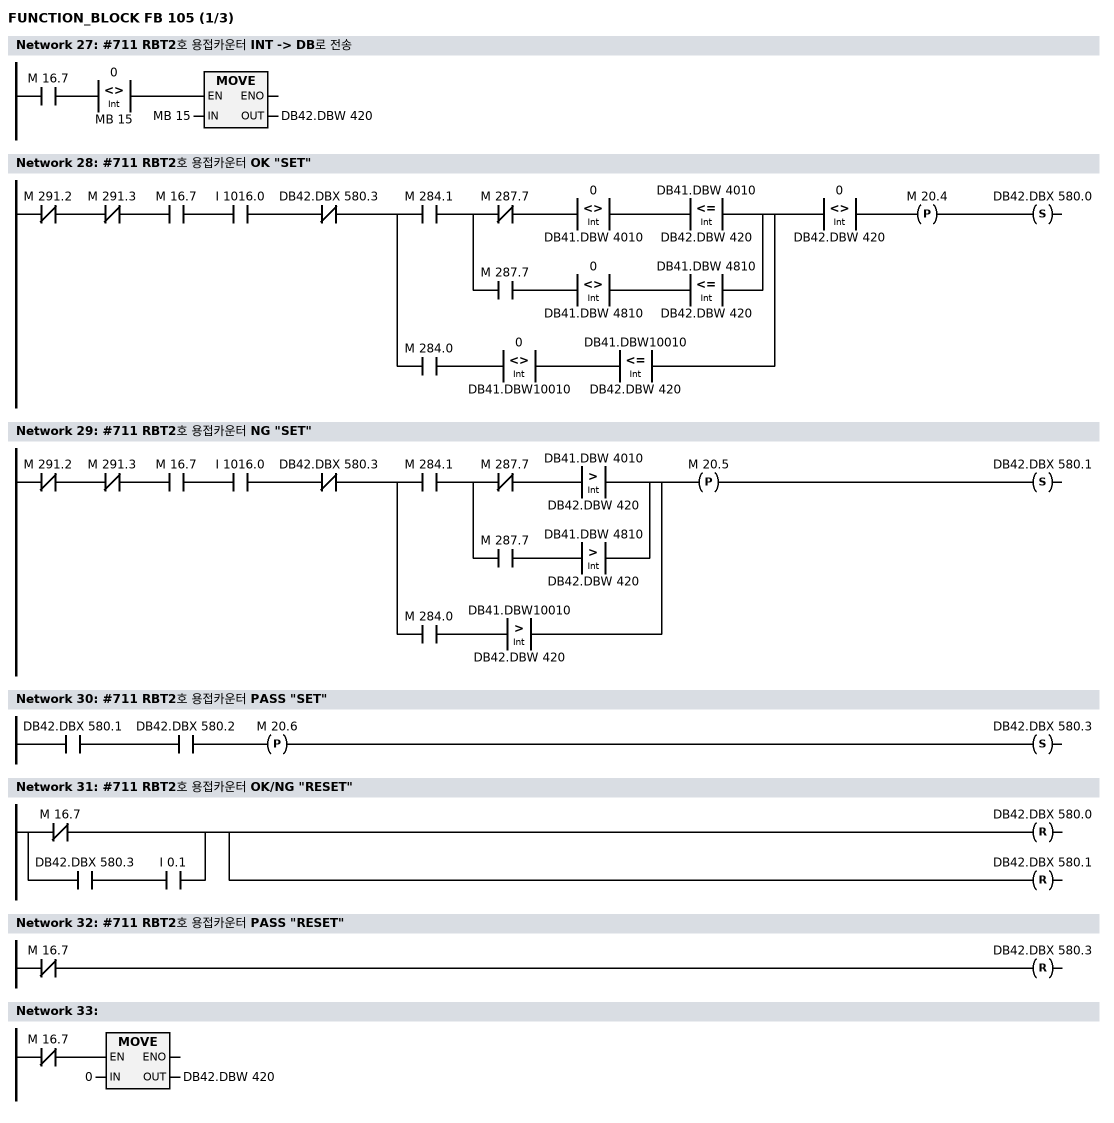

      A     M     16.7;
      A(    ;
      L     0;
      L     MB    15;
      <>I   ;
      )     ;
      JNB   _036;
      L     MB    15;
      T     DB42.DBW  420;
_036: NOP   0;
NETWORK
TITLE =#711 RBT2호 용접카운터 OK "SET"

      AN    M    291.2;
      AN    M    291.3;
      A     M     16.7;
      A     I   1016.0;
      AN    DB42.DBX  580.3;
      A(    ;
      A     M    284.1;
      A(    ;
      AN    M    287.7;
      A(    ;
      L     0;
      L     DB41.DBW 4010;
      <>I   ;
      )     ;
      A(    ;
      L     DB41.DBW 4010;
      L     DB42.DBW  420;
      <=I   ;
      )     ;
      O     ;
      A     M    287.7;
      A(    ;
      L     0;
      L     DB41.DBW 4810;
      <>I   ;
      )     ;
      A(    ;
      L     DB41.DBW 4810;
      L     DB42.DBW  420;
      <=I   ;
      )     ;
      )     ;
      O     ;
      A     M    284.0;
      A(    ;
      L     0;
      L     DB41.DBW10010;
      <>I   ;
      )     ;
      A(    ;
      L     DB41.DBW10010;
      L     DB42.DBW  420;
      <=I   ;
      )     ;
      )     ;
      A(    ;
      L     0;
      L     DB42.DBW  420;
      <>I   ;
      )     ;
      FP    M     20.4;
      S     DB42.DBX  580.0;
NETWORK
TITLE =#711 RBT2호 용접카운터 NG "SET"

      AN    M    291.2;
      AN    M    291.3;
      A     M     16.7;
      A     I   1016.0;
      AN    DB42.DBX  580.3;
      A(    ;
      A     M    284.1;
      A(    ;
      AN    M    287.7;
      A(    ;
      L     DB41.DBW 4010;
      L     DB42.DBW  420;
      >I    ;
      )     ;
      O     ;
      A     M    287.7;
      A(    ;
      L     DB41.DBW 4810;
      L     DB42.DBW  420;
      >I    ;
      )     ;
      )     ;
      O     ;
      A     M    284.0;
      A(    ;
      L     DB41.DBW10010;
      L     DB42.DBW  420;
      >I    ;
      )     ;
      )     ;
      FP    M     20.5;
      S     DB42.DBX  580.1;
NETWORK
TITLE =#711 RBT2호 용접카운터 PASS "SET"

      A     DB42.DBX  580.1;
      A     DB42.DBX  580.2;
      FP    M     20.6;
      S     DB42.DBX  580.3;
NETWORK
TITLE =#711 RBT2호 용접카운터 OK/NG "RESET"

      ON    M     16.7;
      O     ;
      A     DB42.DBX  580.3;
      A     I      0.1;
      R     DB42.DBX  580.0;
      R     DB42.DBX  580.1;
NETWORK
TITLE =#711 RBT2호 용접카운터 PASS "RESET"

      AN    M     16.7;
      R     DB42.DBX  580.3;
NETWORK
TITLE =

      AN    M     16.7;
      JNB   _037;
      L     0;
      T     DB42.DBW  420;
_037: NOP   0;
NETWORK
TITLE =#711 용접DATA 관련(공정 및 차종정보)
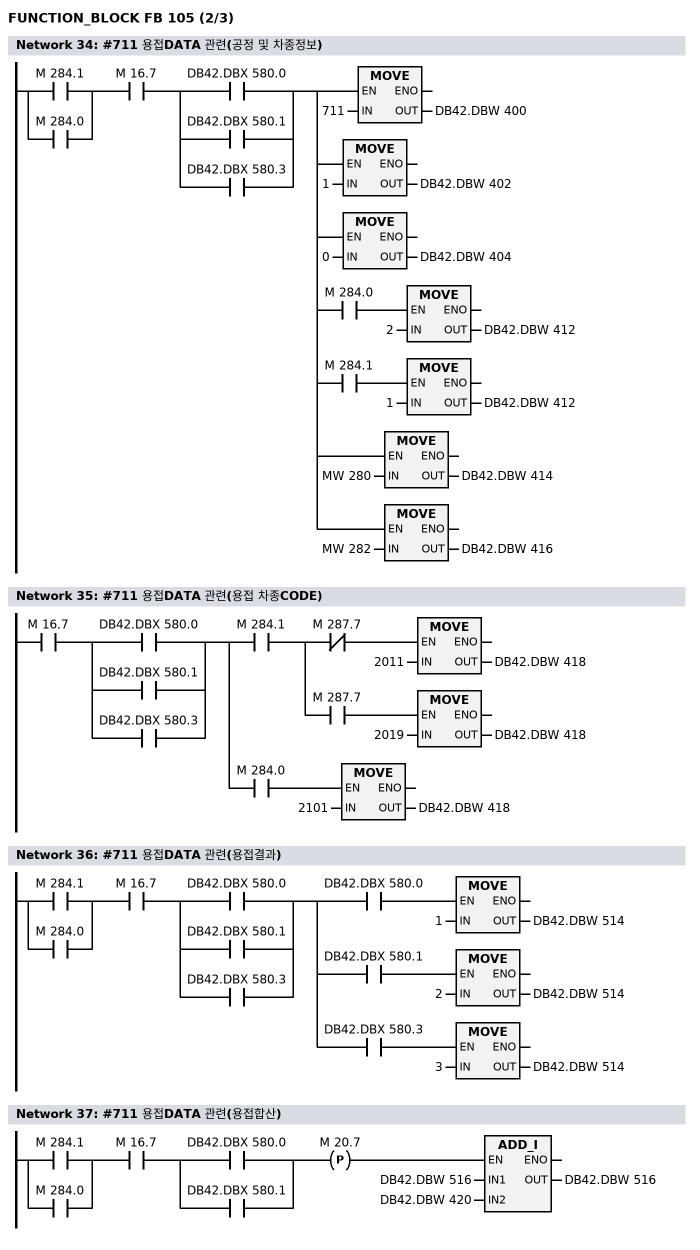

      A(    ;
      O     M    284.1;
      O     M    284.0;
      )     ;
      A     M     16.7;
      A(    ;
      O     DB42.DBX  580.0;
      O     DB42.DBX  580.1;
      O     DB42.DBX  580.3;
      )     ;
      =     L      2.0;
      A     L      2.0;
      JNB   _038;
      L     711;
      T     DB42.DBW  400;
_038: NOP   0;
      A     L      2.0;
      JNB   _039;
      L     1;
      T     DB42.DBW  402;
_039: NOP   0;
      A     L      2.0;
      JNB   _03a;
      L     0;
      T     DB42.DBW  404;
_03a: NOP   0;
      A     L      2.0;
      A     M    284.0;
      JNB   _03b;
      L     2;
      T     DB42.DBW  412;
_03b: NOP   0;
      A     L      2.0;
      A     M    284.1;
      JNB   _03c;
      L     1;
      T     DB42.DBW  412;
_03c: NOP   0;
      A     L      2.0;
      JNB   _03d;
      L     MW   280;
      T     DB42.DBW  414;
_03d: NOP   0;
      A     L      2.0;
      JNB   _03e;
      L     MW   282;
      T     DB42.DBW  416;
_03e: NOP   0;
NETWORK
TITLE =#711 용접DATA 관련(용접 차종CODE)

      A     M     16.7;
      A(    ;
      O     DB42.DBX  580.0;
      O     DB42.DBX  580.1;
      O     DB42.DBX  580.3;
      )     ;
      =     L      2.0;
      A     L      2.0;
      A     M    284.1;
      =     L      2.1;
      A     L      2.1;
      AN    M    287.7;
      JNB   _03f;
      L     2011;
      T     DB42.DBW  418;
_03f: NOP   0;
      A     L      2.1;
      A     M    287.7;
      JNB   _040;
      L     2019;
      T     DB42.DBW  418;
_040: NOP   0;
      A     L      2.0;
      A     M    284.0;
      JNB   _041;
      L     2101;
      T     DB42.DBW  418;
_041: NOP   0;
NETWORK
TITLE =#711 용접DATA 관련(용접결과)

      A(    ;
      O     M    284.1;
      O     M    284.0;
      )     ;
      A     M     16.7;
      A(    ;
      O     DB42.DBX  580.0;
      O     DB42.DBX  580.1;
      O     DB42.DBX  580.3;
      )     ;
      =     L      2.0;
      A     L      2.0;
      A     DB42.DBX  580.0;
      JNB   _042;
      L     1;
      T     DB42.DBW  514;
_042: NOP   0;
      A     L      2.0;
      A     DB42.DBX  580.1;
      JNB   _043;
      L     2;
      T     DB42.DBW  514;
_043: NOP   0;
      A     L      2.0;
      A     DB42.DBX  580.3;
      JNB   _044;
      L     3;
      T     DB42.DBW  514;
_044: NOP   0;
NETWORK
TITLE =#711 용접DATA 관련(용접합산)

      A(    ;
      O     M    284.1;
      O     M    284.0;
      )     ;
      A     M     16.7;
      A(    ;
      O     DB42.DBX  580.0;
      O     DB42.DBX  580.1;
      )     ;
      FP    M     20.7;
      JNB   _045;
      L     DB42.DBW  516;
      L     DB42.DBW  420;
      +I    ;
      T     DB42.DBW  516;
_045: NOP   0;
NETWORK
TITLE =용접누락버퍼로 공정DATA 전송1
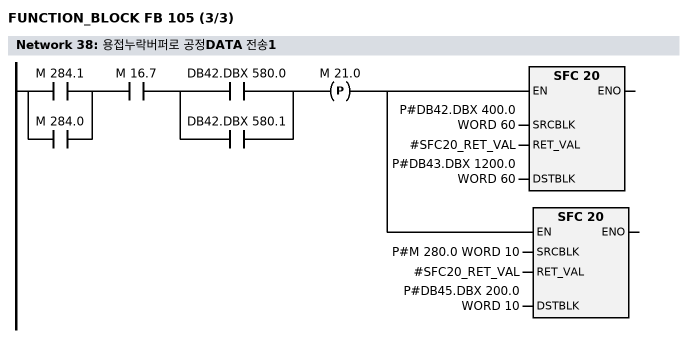

      A(    ;
      O     M    284.1;
      O     M    284.0;
      )     ;
      A     M     16.7;
      A(    ;
      O     DB42.DBX  580.0;
      O     DB42.DBX  580.1;
      )     ;
      FP    M     21.0;
      =     L      2.0;
      A     L      2.0;
      JNB   _046;
      CALL SFC   20 (
           SRCBLK                   := P#DB42.DBX 400.0 WORD 60,
           RET_VAL                  := #SFC20_RET_VAL,
           DSTBLK                   := P#DB43.DBX 1200.0 WORD 60);
_046: NOP   0;
      A     L      2.0;
      JNB   _047;
      CALL SFC   20 (
           SRCBLK                   := P#M 280.0 WORD 10,
           RET_VAL                  := #SFC20_RET_VAL,
           DSTBLK                   := P#DB45.DBX 200.0 WORD 10);
_047: NOP   0;
NETWORK
TITLE =

      AN    M     16.7;
      FP    M     21.1;
      =     L      2.0;
      A(    ;
      A     L      2.0;
      JNB   _048;
      CALL SFC   20 (
           SRCBLK                   := P#DB43.DBX 2160.0 WORD 60,
           RET_VAL                  := #SFC20_RET_VAL,
           DSTBLK                   := P#DB43.DBX 2280.0 WORD 60);
_048: A     BR;
      )     ;
      JNB   _049;
      CALL SFC   20 (
           SRCBLK                   := P#DB43.DBX 2040.0 WORD 60,
           RET_VAL                  := #SFC20_RET_VAL,
           DSTBLK                   := P#DB43.DBX 2160.0 WORD 60);
_049: NOP   0;
      A(    ;
      A     L      2.0;
      JNB   _04a;
      CALL SFC   20 (
           SRCBLK                   := P#DB43.DBX 1920.0 WORD 60,
           RET_VAL                  := #SFC20_RET_VAL,
           DSTBLK                   := P#DB43.DBX 2040.0 WORD 60);
_04a: A     BR;
      )     ;
      JNB   _04b;
      CALL SFC   20 (
           SRCBLK                   := P#DB43.DBX 1800.0 WORD 60,
           RET_VAL                  := #SFC20_RET_VAL,
           DSTBLK                   := P#DB43.DBX 1920.0 WORD 60);
_04b: NOP   0;
      A(    ;
      A     L      2.0;
      JNB   _04c;
      CALL SFC   20 (
           SRCBLK                   := P#DB43.DBX 1680.0 WORD 60,
           RET_VAL                  := #SFC20_RET_VAL,
           DSTBLK                   := P#DB43.DBX 1800.0 WORD 60);
_04c: A     BR;
      )     ;
      JNB   _04d;
      CALL SFC   20 (
           SRCBLK                   := P#DB43.DBX 1560.0 WORD 60,
           RET_VAL                  := #SFC20_RET_VAL,
           DSTBLK                   := P#DB43.DBX 1680.0 WORD 60);
_04d: NOP   0;
      A(    ;
      A     L      2.0;
      JNB   _04e;
      CALL SFC   20 (
           SRCBLK                   := P#DB43.DBX 1440.0 WORD 60,
           RET_VAL                  := #SFC20_RET_VAL,
           DSTBLK                   := P#DB43.DBX 1560.0 WORD 60);
_04e: A     BR;
      )     ;
      JNB   _04f;
      CALL SFC   20 (
           SRCBLK                   := P#DB43.DBX 1320.0 WORD 60,
           RET_VAL                  := #SFC20_RET_VAL,
           DSTBLK                   := P#DB43.DBX 1440.0 WORD 60);
_04f: NOP   0;
      A     L      2.0;
      JNB   _050;
      CALL SFC   20 (
           SRCBLK                   := P#DB43.DBX 1200.0 WORD 60,
           RET_VAL                  := #SFC20_RET_VAL,
           DSTBLK                   := P#DB43.DBX 1320.0 WORD 60);
_050: NOP   0;
      A     L      2.0;
      JNB   _051;
      CALL SFC   21 (
           BVAL                     := P#M 30.0 WORD 1,
           RET_VAL                  := #SFC20_RET_VAL,
           BLK                      := P#DB43.DBX 1200.0 WORD 60);
_051: NOP   0;
      A(    ;
      A     L      2.0;
      JNB   _052;
      CALL SFC   20 (
           SRCBLK                   := P#DB45.DBX 360.0 WORD 10,
           RET_VAL                  := #SFC20_RET_VAL,
           DSTBLK                   := P#DB45.DBX 380.0 WORD 10);
_052: A     BR;
      )     ;
      JNB   _053;
      CALL SFC   20 (
           SRCBLK                   := P#DB45.DBX 340.0 WORD 10,
           RET_VAL                  := #SFC20_RET_VAL,
           DSTBLK                   := P#DB45.DBX 360.0 WORD 10);
_053: NOP   0;
      A(    ;
      A     L      2.0;
      JNB   _054;
      CALL SFC   20 (
           SRCBLK                   := P#DB45.DBX 320.0 WORD 10,
           RET_VAL                  := #SFC20_RET_VAL,
           DSTBLK                   := P#DB45.DBX 340.0 WORD 10);
_054: A     BR;
      )     ;
      JNB   _055;
      CALL SFC   20 (
           SRCBLK                   := P#DB45.DBX 300.0 WORD 10,
           RET_VAL                  := #SFC20_RET_VAL,
           DSTBLK                   := P#DB45.DBX 320.0 WORD 10);
_055: NOP   0;
      A(    ;
      A     L      2.0;
      JNB   _056;
      CALL SFC   20 (
           SRCBLK                   := P#DB45.DBX 280.0 WORD 10,
           RET_VAL                  := #SFC20_RET_VAL,
           DSTBLK                   := P#DB45.DBX 300.0 WORD 10);
_056: A     BR;
      )     ;
      JNB   _057;
      CALL SFC   20 (
           SRCBLK                   := P#DB45.DBX 260.0 WORD 10,
           RET_VAL                  := #SFC20_RET_VAL,
           DSTBLK                   := P#DB45.DBX 280.0 WORD 10);
_057: NOP   0;
      A(    ;
      A     L      2.0;
      JNB   _058;
      CALL SFC   20 (
           SRCBLK                   := P#DB45.DBX 240.0 WORD 10,
           RET_VAL                  := #SFC20_RET_VAL,
           DSTBLK                   := P#DB45.DBX 260.0 WORD 10);
_058: A     BR;
      )     ;
      JNB   _059;
      CALL SFC   20 (
           SRCBLK                   := P#DB45.DBX 220.0 WORD 10,
           RET_VAL                  := #SFC20_RET_VAL,
           DSTBLK                   := P#DB45.DBX 240.0 WORD 10);
_059: NOP   0;
      A     L      2.0;
      JNB   _05a;
      CALL SFC   20 (
           SRCBLK                   := P#DB45.DBX 200.0 WORD 10,
           RET_VAL                  := #SFC20_RET_VAL,
           DSTBLK                   := P#DB45.DBX 220.0 WORD 10);
_05a: NOP   0;
      A     L      2.0;
      JNB   _05b;
      CALL SFC   21 (
           BVAL                     := P#M 30.0 WORD 1,
           RET_VAL                  := #SFC20_RET_VAL,
           BLK                      := P#DB45.DBX 200.0 WORD 10);
_05b: NOP   0;
NETWORK
TITLE =용접누락버퍼로 공정DATA 전송1
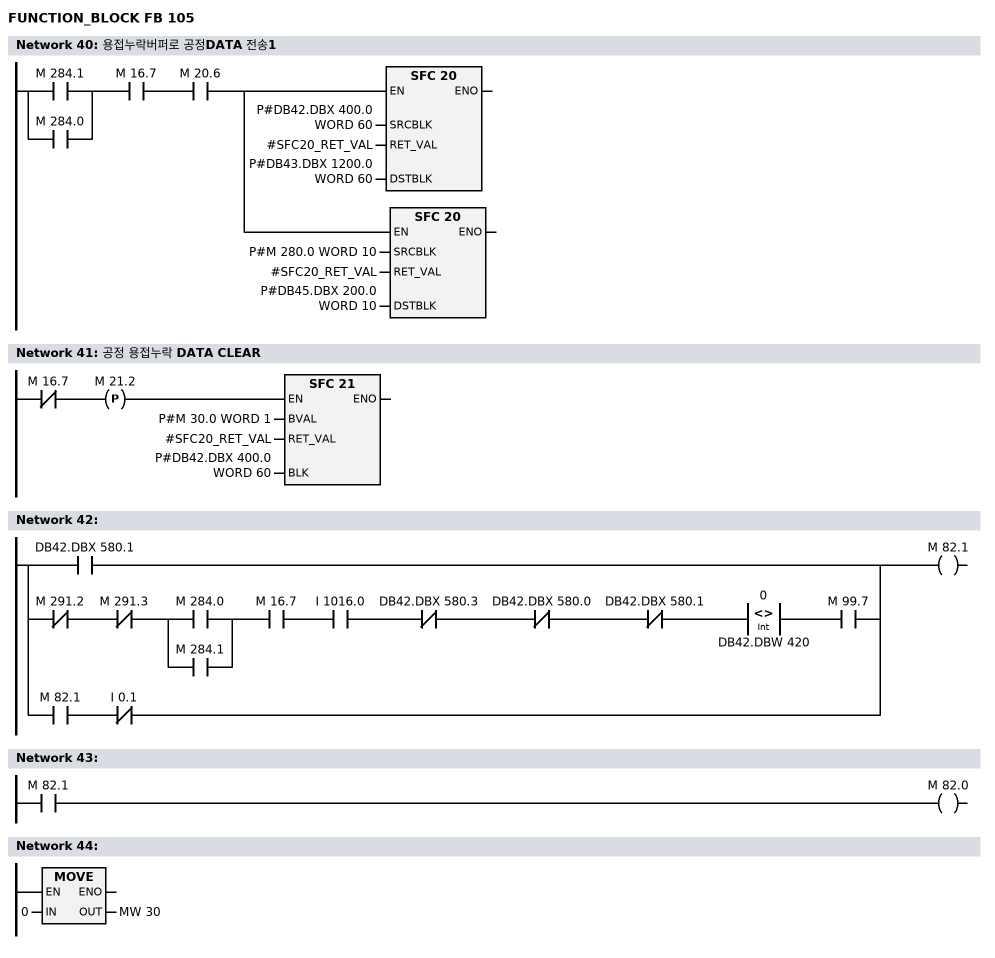

      A(    ;
      O     M    284.1;
      O     M    284.0;
      )     ;
      A     M     16.7;
      A     M     20.6;
      =     L      2.0;
      A     L      2.0;
      JNB   _05c;
      CALL SFC   20 (
           SRCBLK                   := P#DB42.DBX 400.0 WORD 60,
           RET_VAL                  := #SFC20_RET_VAL,
           DSTBLK                   := P#DB43.DBX 1200.0 WORD 60);
_05c: NOP   0;
      A     L      2.0;
      JNB   _05d;
      CALL SFC   20 (
           SRCBLK                   := P#M 280.0 WORD 10,
           RET_VAL                  := #SFC20_RET_VAL,
           DSTBLK                   := P#DB45.DBX 200.0 WORD 10);
_05d: NOP   0;
NETWORK
TITLE =공정 용접누락 DATA CLEAR

      AN    M     16.7;
      FP    M     21.2;
      JNB   _05e;
      CALL SFC   21 (
           BVAL                     := P#M 30.0 WORD 1,
           RET_VAL                  := #SFC20_RET_VAL,
           BLK                      := P#DB42.DBX 400.0 WORD 60);
_05e: NOP   0;
NETWORK
TITLE =

      O     DB42.DBX  580.1;
      O     ;
      AN    M    291.2;
      AN    M    291.3;
      A(    ;
      O     M    284.0;
      O     M    284.1;
      )     ;
      A     M     16.7;
      A     I   1016.0;
      AN    DB42.DBX  580.3;
      AN    DB42.DBX  580.0;
      AN    DB42.DBX  580.1;
      A(    ;
      L     0;
      L     DB42.DBW  420;
      <>I   ;
      )     ;
      A     M     99.7;
      O     ;
      A     M     82.1;
      AN    I      0.1;
      =     M     82.1;
NETWORK
TITLE =

      A     M     82.1;
      =     M     82.0;
NETWORK
TITLE =

      L     0;
      T     MW    30;
      NOP   0;
END_FUNCTION_BLOCK

DATA_BLOCK DB 105
TITLE =
VERSION : 0.0

 FB 105
BEGIN
   S711A_RBT1_WELD_OK_PLS := FALSE;
   S711A_RBT1_WELD_NG_PLS := FALSE;
   S711A_RBT1_WELD_PASS_PLS := FALSE;
   S711A_CHECK_SUM_PLS := FALSE;
   S711A_WELD_DATA_MOV_BUFF := FALSE;
   MW_0_BUFF[0] := W#16#0;
   MW_0_BUFF[1] := W#16#0;
   MW_0_BUFF[2] := W#16#0;
   MW_0_BUFF[3] := W#16#0;
   MW_0_BUFF[4] := W#16#0;
   MW_0_BUFF[5] := W#16#0;
   MW_0_BUFF[6] := W#16#0;
   MW_0_BUFF[7] := W#16#0;
   MW_0_BUFF[8] := W#16#0;
   MW_0_BUFF[9] := W#16#0;
   MW_0_BUFF[10] := W#16#0;
   MW_0_BUFF[11] := W#16#0;
   MW_0_BUFF[12] := W#16#0;
   MW_0_BUFF[13] := W#16#0;
   MW_0_BUFF[14] := W#16#0;
   MW_0_BUFF[15] := W#16#0;
   MW_0_BUFF[16] := W#16#0;
   MW_0_BUFF[17] := W#16#0;
   MW_0_BUFF[18] := W#16#0;
   MW_0_BUFF[19] := W#16#0;
   MW_0_BUFF[20] := W#16#0;
   MW_0_BUFF[21] := W#16#0;
   MW_0_BUFF[22] := W#16#0;
   MW_0_BUFF[23] := W#16#0;
   MW_0_BUFF[24] := W#16#0;
   MW_0_BUFF[25] := W#16#0;
   MW_0_BUFF[26] := W#16#0;
   MW_0_BUFF[27] := W#16#0;
   MW_0_BUFF[28] := W#16#0;
   MW_0_BUFF[29] := W#16#0;
   MW_0_BUFF[30] := W#16#0;
   MW_0_BUFF[31] := W#16#0;
   MW_0_BUFF[32] := W#16#0;
   MW_0_BUFF[33] := W#16#0;
   MW_0_BUFF[34] := W#16#0;
   MW_0_BUFF[35] := W#16#0;
   MW_0_BUFF[36] := W#16#0;
   MW_0_BUFF[37] := W#16#0;
   MW_0_BUFF[38] := W#16#0;
   MW_0_BUFF[39] := W#16#0;
   MW_0_BUFF[40] := W#16#0;
   MW_0_BUFF[41] := W#16#0;
   MW_0_BUFF[42] := W#16#0;
   MW_0_BUFF[43] := W#16#0;
   MW_0_BUFF[44] := W#16#0;
   MW_0_BUFF[45] := W#16#0;
   MW_0_BUFF[46] := W#16#0;
   MW_0_BUFF[47] := W#16#0;
   MW_0_BUFF[48] := W#16#0;
   MW_0_BUFF[49] := W#16#0;
   MW_0_BUFF[50] := W#16#0;
   MW_0_BUFF[51] := W#16#0;
   MW_0_BUFF[52] := W#16#0;
   MW_0_BUFF[53] := W#16#0;
   MW_0_BUFF[54] := W#16#0;
   MW_0_BUFF[55] := W#16#0;
   MW_0_BUFF[56] := W#16#0;
   MW_0_BUFF[57] := W#16#0;
   MW_0_BUFF[58] := W#16#0;
   MW_0_BUFF[59] := W#16#0;
   PLS1 := FALSE;
   PLS2 := FALSE;
END_DATA_BLOCK

FUNCTION_BLOCK FB 106
TITLE =
VERSION : 0.1


VAR
  CAR_TYPE_MODIFY : FB 470;
  SFC20_RET_VAL : INT ;
  HMI_CAR_TYPE_V2 : FB 512;
  S6_HMI_CAR_TYPE_V2 : FB 512;
  S6_CAR_TYPE_MODIFY : FB 470;
  S486RH_CARTYPE : FB 512;
  S486LH_CARTYPE : FB 512;
  S711_CARTYPE : FB 512;
  S711R1_R2_CARTYPE : FB 512;
  S711A_FAC_CARTYPE : FB 512;
  S711AB_KEY_CARTYPE : FB 512;
  S711A_R1_CARTYPE : FB 512;
  S711_IDLE_CARTYPE : FB 512;
END_VAR
VAR_TEMP
  SFC21_RET_VAL : INT ;
END_VAR
BEGIN
NETWORK
TITLE =
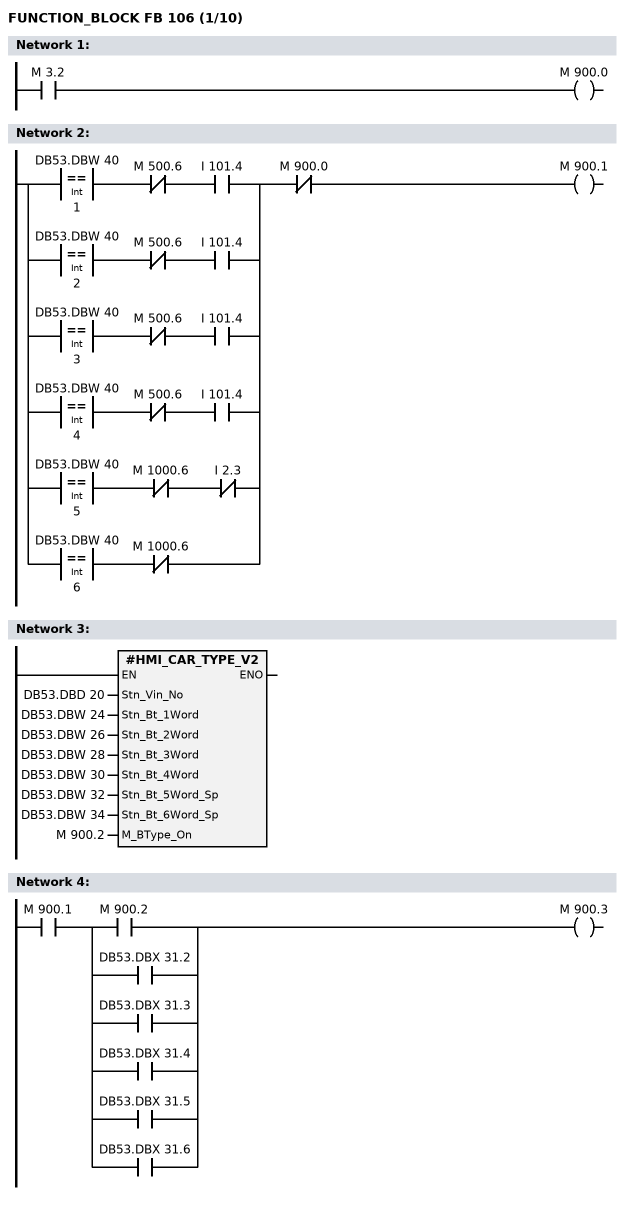

      A     M      3.2;
      =     M    900.0;
NETWORK
TITLE =

      A(    ;
      A(    ;
      L     DB53.DBW   40;
      L     1;
      ==I   ;
      )     ;
      AN    M    500.6;
      A     I    101.4;
      O     ;
      A(    ;
      L     DB53.DBW   40;
      L     2;
      ==I   ;
      )     ;
      AN    M    500.6;
      A     I    101.4;
      O     ;
      A(    ;
      L     DB53.DBW   40;
      L     3;
      ==I   ;
      )     ;
      AN    M    500.6;
      A     I    101.4;
      O     ;
      A(    ;
      L     DB53.DBW   40;
      L     4;
      ==I   ;
      )     ;
      AN    M    500.6;
      A     I    101.4;
      O     ;
      A(    ;
      L     DB53.DBW   40;
      L     5;
      ==I   ;
      )     ;
      AN    M   1000.6;
      AN    I      2.3;
      O     ;
      A(    ;
      L     DB53.DBW   40;
      L     6;
      ==I   ;
      )     ;
      AN    M   1000.6;
      )     ;
      AN    M    900.0;
      =     M    900.1;
NETWORK
TITLE =

      CALL #HMI_CAR_TYPE_V2 (
           Stn_Vin_No               := DB53.DBD   20,
           Stn_Bt_1Word             := DB53.DBW   24,
           Stn_Bt_2Word             := DB53.DBW   26,
           Stn_Bt_3Word             := DB53.DBW   28,
           Stn_Bt_4Word             := DB53.DBW   30,
           Stn_Bt_5Word_Sp          := DB53.DBW   32,
           Stn_Bt_6Word_Sp          := DB53.DBW   34,
           M_BType_On               := M    900.2);

      NOP   0;
NETWORK
TITLE =

      A     M    900.1;
      A(    ;
      O     M    900.2;
      O     DB53.DBX   31.2;
      O     DB53.DBX   31.3;
      O     DB53.DBX   31.4;
      O     DB53.DBX   31.5;
      O     DB53.DBX   31.6;
      )     ;
      =     M    900.3;
NETWORK
TITLE =
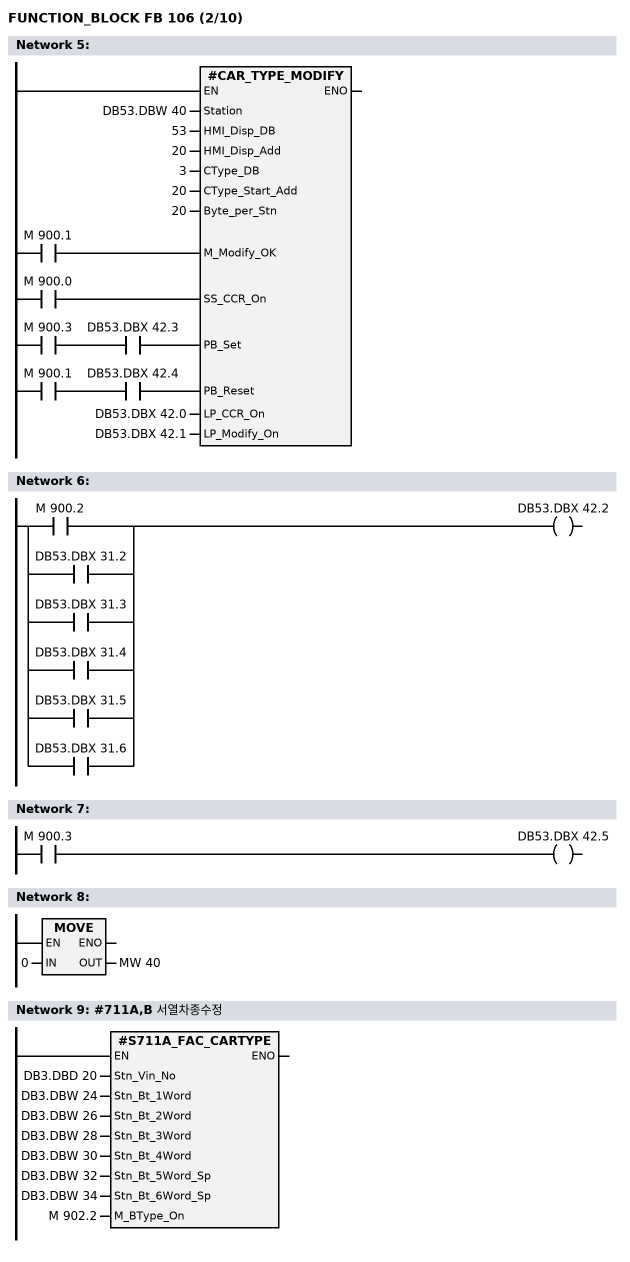

      A     M    900.1;
      =     L      2.0;
      BLD   103;
      A     M    900.0;
      =     L      2.1;
      BLD   103;
      A     M    900.3;
      A     DB53.DBX   42.3;
      =     L      2.2;
      BLD   103;
      A     M    900.1;
      A     DB53.DBX   42.4;
      =     L      2.3;
      BLD   103;
      CALL #CAR_TYPE_MODIFY (
           Station                  := DB53.DBW   40,
           HMI_Disp_DB              := 53,
           HMI_Disp_Add             := 20,
           CType_DB                 := 3,
           CType_Start_Add          := 20,
           Byte_per_Stn             := 20,
           M_Modify_OK              := L      2.0,
           SS_CCR_On                := L      2.1,
           PB_Set                   := L      2.2,
           PB_Reset                 := L      2.3,
           LP_CCR_On                := DB53.DBX   42.0,
           LP_Modify_On             := DB53.DBX   42.1);
      NOP   0;
NETWORK
TITLE =

      O     M    900.2;
      O     DB53.DBX   31.2;
      O     DB53.DBX   31.3;
      O     DB53.DBX   31.4;
      O     DB53.DBX   31.5;
      O     DB53.DBX   31.6;
      =     DB53.DBX   42.2;
NETWORK
TITLE =

      A     M    900.3;
      =     DB53.DBX   42.5;
NETWORK
TITLE =

      L     0;
      T     MW    40;
      NOP   0;
NETWORK
TITLE =#711A,B 서열차종수정

      CALL #S711A_FAC_CARTYPE (
           Stn_Vin_No               := DB3.DBD   20,
           Stn_Bt_1Word             := DB3.DBW   24,
           Stn_Bt_2Word             := DB3.DBW   26,
           Stn_Bt_3Word             := DB3.DBW   28,
           Stn_Bt_4Word             := DB3.DBW   30,
           Stn_Bt_5Word_Sp          := DB3.DBW   32,
           Stn_Bt_6Word_Sp          := DB3.DBW   34,
           M_BType_On               := M    902.2);

      NOP   0;
NETWORK
TITLE =#711A,B 차종수정
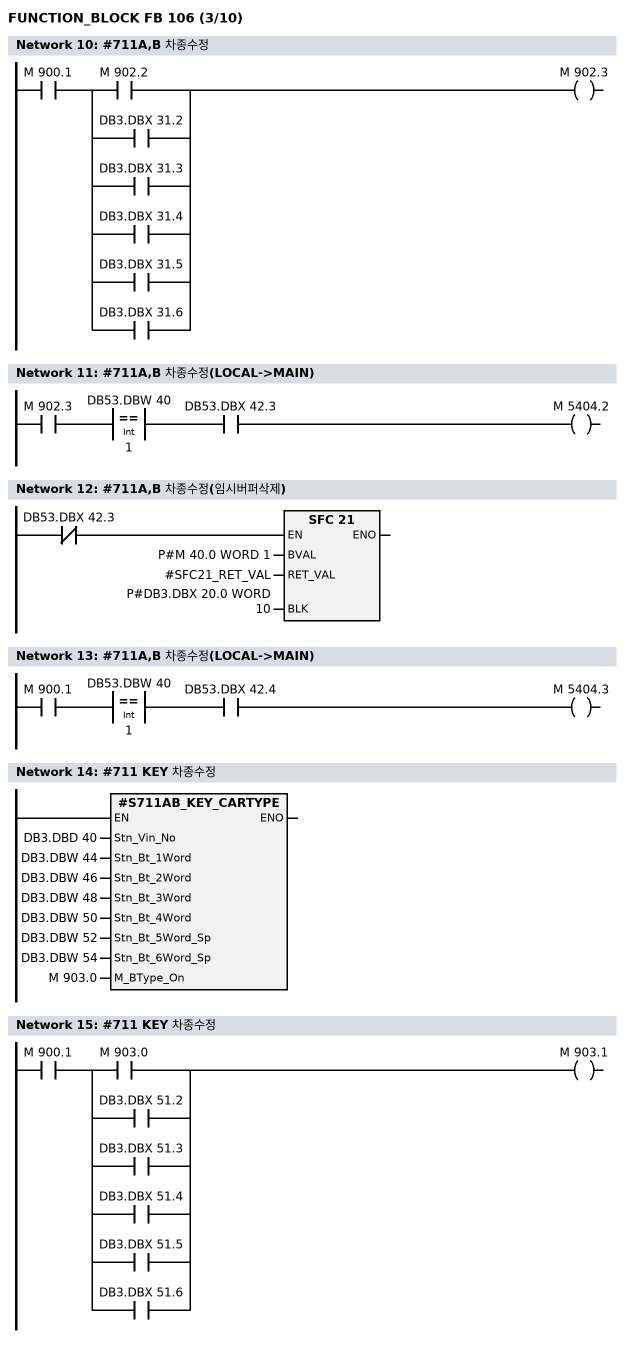

      A     M    900.1;
      A(    ;
      O     M    902.2;
      O     DB3.DBX   31.2;
      O     DB3.DBX   31.3;
      O     DB3.DBX   31.4;
      O     DB3.DBX   31.5;
      O     DB3.DBX   31.6;
      )     ;
      =     M    902.3;
NETWORK
TITLE =#711A,B 차종수정(LOCAL->MAIN)

      A     M    902.3;
      A(    ;
      L     DB53.DBW   40;
      L     1;
      ==I   ;
      )     ;
      A     DB53.DBX   42.3;
      =     M   5404.2;
NETWORK
TITLE =#711A,B 차종수정(임시버퍼삭제)

      AN    DB53.DBX   42.3;
      JNB   _001;
      CALL SFC   21 (
           BVAL                     := P#M 40.0 WORD 1,
           RET_VAL                  := #SFC21_RET_VAL,
           BLK                      := P#DB3.DBX 20.0 WORD 10);
_001: NOP   0;
NETWORK
TITLE =#711A,B 차종수정(LOCAL->MAIN)

      A     M    900.1;
      A(    ;
      L     DB53.DBW   40;
      L     1;
      ==I   ;
      )     ;
      A     DB53.DBX   42.4;
      =     M   5404.3;
NETWORK
TITLE =#711 KEY 차종수정

      CALL #S711AB_KEY_CARTYPE (
           Stn_Vin_No               := DB3.DBD   40,
           Stn_Bt_1Word             := DB3.DBW   44,
           Stn_Bt_2Word             := DB3.DBW   46,
           Stn_Bt_3Word             := DB3.DBW   48,
           Stn_Bt_4Word             := DB3.DBW   50,
           Stn_Bt_5Word_Sp          := DB3.DBW   52,
           Stn_Bt_6Word_Sp          := DB3.DBW   54,
           M_BType_On               := M    903.0);

      NOP   0;
NETWORK
TITLE =#711 KEY 차종수정

      A     M    900.1;
      A(    ;
      O     M    903.0;
      O     DB3.DBX   51.2;
      O     DB3.DBX   51.3;
      O     DB3.DBX   51.4;
      O     DB3.DBX   51.5;
      O     DB3.DBX   51.6;
      )     ;
      =     M    903.1;
NETWORK
TITLE =#711 KEY 차종수정
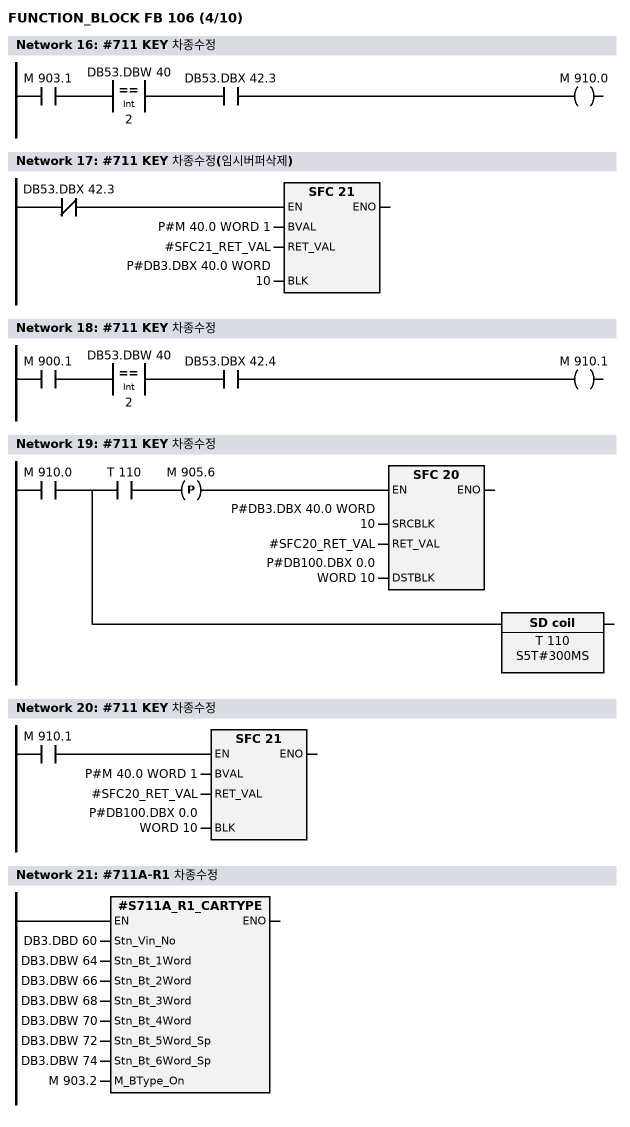

      A     M    903.1;
      A(    ;
      L     DB53.DBW   40;
      L     2;
      ==I   ;
      )     ;
      A     DB53.DBX   42.3;
      =     M    910.0;
NETWORK
TITLE =#711 KEY 차종수정(임시버퍼삭제)

      AN    DB53.DBX   42.3;
      JNB   _002;
      CALL SFC   21 (
           BVAL                     := P#M 40.0 WORD 1,
           RET_VAL                  := #SFC21_RET_VAL,
           BLK                      := P#DB3.DBX 40.0 WORD 10);
_002: NOP   0;
NETWORK
TITLE =#711 KEY 차종수정

      A     M    900.1;
      A(    ;
      L     DB53.DBW   40;
      L     2;
      ==I   ;
      )     ;
      A     DB53.DBX   42.4;
      =     M    910.1;
NETWORK
TITLE =#711 KEY 차종수정

      A     M    910.0;
      =     L      2.0;
      A     L      2.0;
      A     T    110;
      FP    M    905.6;
      JNB   _003;
      CALL SFC   20 (
           SRCBLK                   := P#DB3.DBX 40.0 WORD 10,
           RET_VAL                  := #SFC20_RET_VAL,
           DSTBLK                   := P#DB100.DBX 0.0 WORD 10);
_003: NOP   0;
      A     L      2.0;
      BLD   102;
      L     S5T#300MS;
      SD    T    110;
NETWORK
TITLE =#711 KEY 차종수정

      A     M    910.1;
      JNB   _004;
      CALL SFC   21 (
           BVAL                     := P#M 40.0 WORD 1,
           RET_VAL                  := #SFC20_RET_VAL,
           BLK                      := P#DB100.DBX 0.0 WORD 10);
_004: NOP   0;
NETWORK
TITLE =#711A-R1 차종수정

      CALL #S711A_R1_CARTYPE (
           Stn_Vin_No               := DB3.DBD   60,
           Stn_Bt_1Word             := DB3.DBW   64,
           Stn_Bt_2Word             := DB3.DBW   66,
           Stn_Bt_3Word             := DB3.DBW   68,
           Stn_Bt_4Word             := DB3.DBW   70,
           Stn_Bt_5Word_Sp          := DB3.DBW   72,
           Stn_Bt_6Word_Sp          := DB3.DBW   74,
           M_BType_On               := M    903.2);

      NOP   0;
NETWORK
TITLE =#711A-R1 차종수정
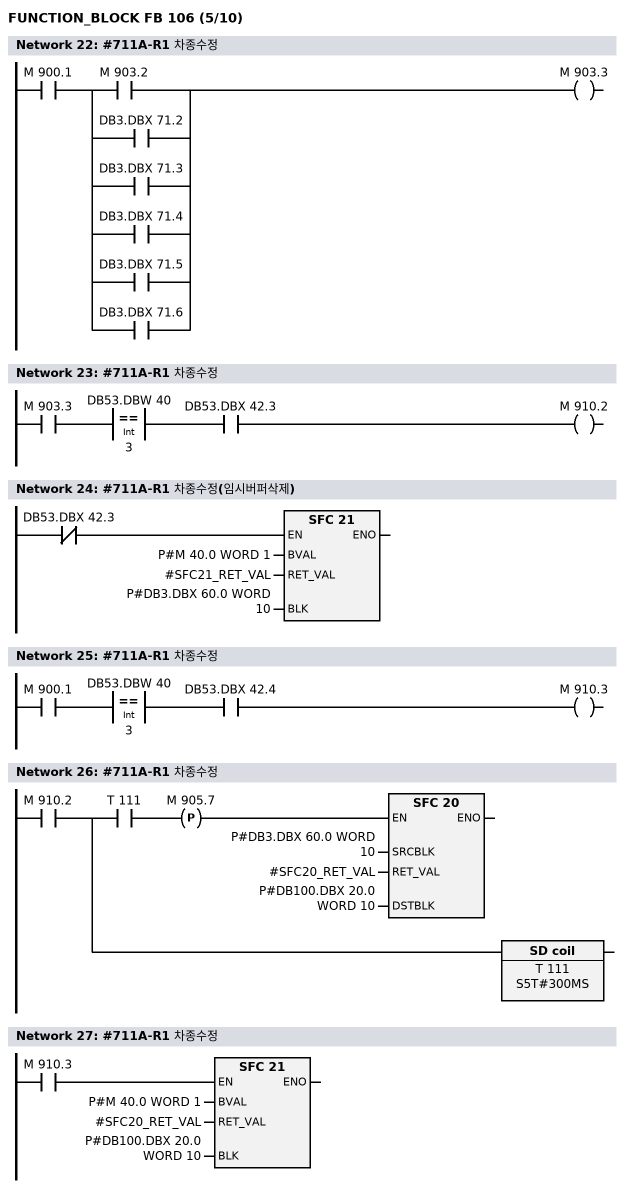

      A     M    900.1;
      A(    ;
      O     M    903.2;
      O     DB3.DBX   71.2;
      O     DB3.DBX   71.3;
      O     DB3.DBX   71.4;
      O     DB3.DBX   71.5;
      O     DB3.DBX   71.6;
      )     ;
      =     M    903.3;
NETWORK
TITLE =#711A-R1 차종수정

      A     M    903.3;
      A(    ;
      L     DB53.DBW   40;
      L     3;
      ==I   ;
      )     ;
      A     DB53.DBX   42.3;
      =     M    910.2;
NETWORK
TITLE =#711A-R1 차종수정(임시버퍼삭제)

      AN    DB53.DBX   42.3;
      JNB   _005;
      CALL SFC   21 (
           BVAL                     := P#M 40.0 WORD 1,
           RET_VAL                  := #SFC21_RET_VAL,
           BLK                      := P#DB3.DBX 60.0 WORD 10);
_005: NOP   0;
NETWORK
TITLE =#711A-R1 차종수정

      A     M    900.1;
      A(    ;
      L     DB53.DBW   40;
      L     3;
      ==I   ;
      )     ;
      A     DB53.DBX   42.4;
      =     M    910.3;
NETWORK
TITLE =#711A-R1 차종수정

      A     M    910.2;
      =     L      2.0;
      A     L      2.0;
      A     T    111;
      FP    M    905.7;
      JNB   _006;
      CALL SFC   20 (
           SRCBLK                   := P#DB3.DBX 60.0 WORD 10,
           RET_VAL                  := #SFC20_RET_VAL,
           DSTBLK                   := P#DB100.DBX 20.0 WORD 10);
_006: NOP   0;
      A     L      2.0;
      BLD   102;
      L     S5T#300MS;
      SD    T    111;
NETWORK
TITLE =#711A-R1 차종수정

      A     M    910.3;
      JNB   _007;
      CALL SFC   21 (
           BVAL                     := P#M 40.0 WORD 1,
           RET_VAL                  := #SFC20_RET_VAL,
           BLK                      := P#DB100.DBX 20.0 WORD 10);
_007: NOP   0;
NETWORK
TITLE =#711 IDLE 차종수정
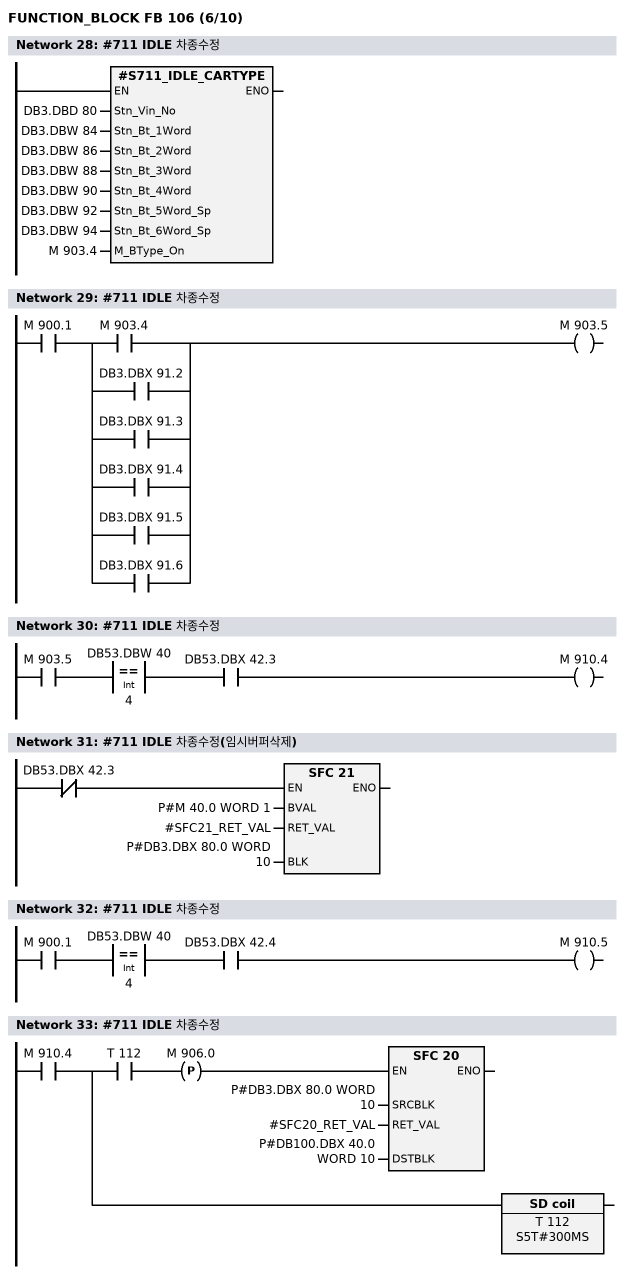

      CALL #S711_IDLE_CARTYPE (
           Stn_Vin_No               := DB3.DBD   80,
           Stn_Bt_1Word             := DB3.DBW   84,
           Stn_Bt_2Word             := DB3.DBW   86,
           Stn_Bt_3Word             := DB3.DBW   88,
           Stn_Bt_4Word             := DB3.DBW   90,
           Stn_Bt_5Word_Sp          := DB3.DBW   92,
           Stn_Bt_6Word_Sp          := DB3.DBW   94,
           M_BType_On               := M    903.4);

      NOP   0;
NETWORK
TITLE =#711 IDLE 차종수정

      A     M    900.1;
      A(    ;
      O     M    903.4;
      O     DB3.DBX   91.2;
      O     DB3.DBX   91.3;
      O     DB3.DBX   91.4;
      O     DB3.DBX   91.5;
      O     DB3.DBX   91.6;
      )     ;
      =     M    903.5;
NETWORK
TITLE =#711 IDLE 차종수정

      A     M    903.5;
      A(    ;
      L     DB53.DBW   40;
      L     4;
      ==I   ;
      )     ;
      A     DB53.DBX   42.3;
      =     M    910.4;
NETWORK
TITLE =#711 IDLE 차종수정(임시버퍼삭제)

      AN    DB53.DBX   42.3;
      JNB   _008;
      CALL SFC   21 (
           BVAL                     := P#M 40.0 WORD 1,
           RET_VAL                  := #SFC21_RET_VAL,
           BLK                      := P#DB3.DBX 80.0 WORD 10);
_008: NOP   0;
NETWORK
TITLE =#711 IDLE 차종수정

      A     M    900.1;
      A(    ;
      L     DB53.DBW   40;
      L     4;
      ==I   ;
      )     ;
      A     DB53.DBX   42.4;
      =     M    910.5;
NETWORK
TITLE =#711 IDLE 차종수정

      A     M    910.4;
      =     L      2.0;
      A     L      2.0;
      A     T    112;
      FP    M    906.0;
      JNB   _009;
      CALL SFC   20 (
           SRCBLK                   := P#DB3.DBX 80.0 WORD 10,
           RET_VAL                  := #SFC20_RET_VAL,
           DSTBLK                   := P#DB100.DBX 40.0 WORD 10);
_009: NOP   0;
      A     L      2.0;
      BLD   102;
      L     S5T#300MS;
      SD    T    112;
NETWORK
TITLE =#711 KEY 차종수정
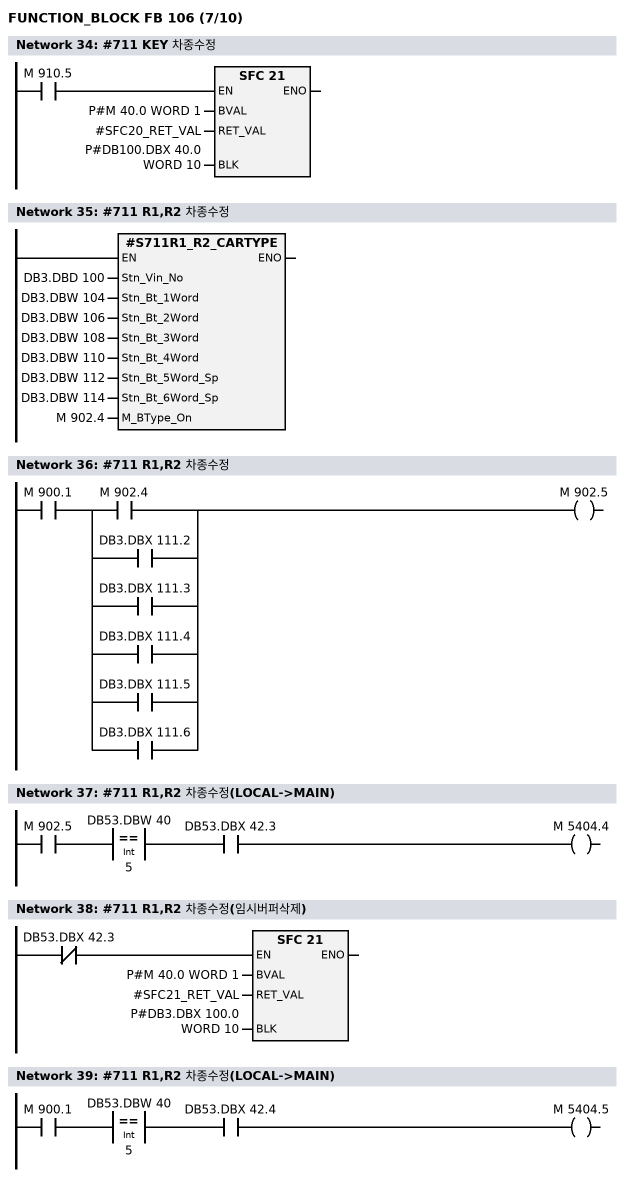

      A     M    910.5;
      JNB   _00a;
      CALL SFC   21 (
           BVAL                     := P#M 40.0 WORD 1,
           RET_VAL                  := #SFC20_RET_VAL,
           BLK                      := P#DB100.DBX 40.0 WORD 10);
_00a: NOP   0;
NETWORK
TITLE =#711 R1,R2 차종수정

      CALL #S711R1_R2_CARTYPE (
           Stn_Vin_No               := DB3.DBD  100,
           Stn_Bt_1Word             := DB3.DBW  104,
           Stn_Bt_2Word             := DB3.DBW  106,
           Stn_Bt_3Word             := DB3.DBW  108,
           Stn_Bt_4Word             := DB3.DBW  110,
           Stn_Bt_5Word_Sp          := DB3.DBW  112,
           Stn_Bt_6Word_Sp          := DB3.DBW  114,
           M_BType_On               := M    902.4);

      NOP   0;
NETWORK
TITLE =#711 R1,R2 차종수정

      A     M    900.1;
      A(    ;
      O     M    902.4;
      O     DB3.DBX  111.2;
      O     DB3.DBX  111.3;
      O     DB3.DBX  111.4;
      O     DB3.DBX  111.5;
      O     DB3.DBX  111.6;
      )     ;
      =     M    902.5;
NETWORK
TITLE =#711 R1,R2 차종수정(LOCAL->MAIN)

      A     M    902.5;
      A(    ;
      L     DB53.DBW   40;
      L     5;
      ==I   ;
      )     ;
      A     DB53.DBX   42.3;
      =     M   5404.4;
NETWORK
TITLE =#711 R1,R2 차종수정(임시버퍼삭제)

      AN    DB53.DBX   42.3;
      JNB   _00b;
      CALL SFC   21 (
           BVAL                     := P#M 40.0 WORD 1,
           RET_VAL                  := #SFC21_RET_VAL,
           BLK                      := P#DB3.DBX 100.0 WORD 10);
_00b: NOP   0;
NETWORK
TITLE =#711 R1,R2 차종수정(LOCAL->MAIN)

      A     M    900.1;
      A(    ;
      L     DB53.DBW   40;
      L     5;
      ==I   ;
      )     ;
      A     DB53.DBX   42.4;
      =     M   5404.5;
NETWORK
TITLE =#711 차종수정
